   VAR_IN_OUT
      iqUDT_EquipmentControl : "UDT_EquipmentControl";   // Equipment control structure
      iqUDT_ConveyorInterface : "UDT_ConveyorInterface";   // Interface structure
   END_VAR

   VAR
      sx_EncoderFault { ExternalAccessible := 'False'; ExternalVisible := 'False'; ExternalWritable := 'False'} : Bool;   // When TRUE encoder fault is active
      slr_ActualDelayTime { ExternalAccessible := 'False'; ExternalVisible := 'False'; ExternalWritable := 'False'} : LReal;   // Actual delay time [ms]
   END_VAR

   VAR CONSTANT
      cudi_EncoderFaultDelayTime : UDInt := 5000;   // Time after which the encoder fault is activated
   END_VAR


BEGIN
	(*
	----------------------------------------------------------------------------------------

	Version history:
	Date        | Version   | Author        | Remark
	----------------------------------------------------------------------------------------
	19/07/2022  | 0.1       | M.Kurpiers    | first release MHS TIA 16.0
	21/02/2023  | 4.0       | F.Baten       | 4.0 Release TIA 17.5
	*)

	REGION 1 - Reset encoder error

	    IF #iqUDT_EquipmentControl.Command.Reset OR #iqUDT_ConveyorInterface.InternalErrorReset THEN
	        #sx_EncoderFault := FALSE;
	    END_IF;

	END_REGION

	REGION 2 - Set encoder error

	    IF #iqUDT_ConveyorInterface.ActualSpeed > 0
	        AND NOT #ix_EncoderPulses
	        AND NOT #iqUDT_ConveyorInterface.ManualModeActive THEN

	        #slr_ActualDelayTime += "DB_Memory".PrevCycleTime;

	        IF #slr_ActualDelayTime >= #cudi_EncoderFaultDelayTime THEN
	            #sx_EncoderFault := TRUE;
	        END_IF;
	    ELSE
	        #slr_ActualDelayTime := 0;
	    END_IF;

	    #iqUDT_ConveyorInterface.InternalErrorEncoder := #sx_EncoderFault;

	END_REGION

	REGION 3 - Status

	    #qUDT_HMIStatus.Fault := #sx_EncoderFault;

	END_REGION


END_FUNCTION_BLOCK

FUNCTION_BLOCK "FB_Valve"
TITLE = Single ended Valve Control and monitor
{ S7_Optimized_Access := 'TRUE' }
AUTHOR : 'I.Ajram'
VERSION : 0.1
   VAR_INPUT
      iUDT_Configuration { ExternalAccessible := 'False'; ExternalVisible := 'False'; ExternalWritable := 'False'} : "UDT_ValveConfiguration";   // Valve configuration
      ix_Open { ExternalAccessible := 'False'; ExternalVisible := 'False'; ExternalWritable := 'False'} : Bool;   // Open command (Hold if ControlMode = 1, pulse if ControlMode = 2)
      ix_Close { ExternalAccessible := 'False'; ExternalVisible := 'False'; ExternalWritable := 'False'} : Bool;   // Close command (Not used if ControlMode = 1, pulse if ControlMode = 2)
      ix_IsOpened { ExternalAccessible := 'False'; ExternalVisible := 'False'; ExternalWritable := 'False'} : Bool;   // Feedback Signal ( Not used if #iqUDT_SEVConfiguration.IsOpenFeedBackExist is FALSE)
      ix_IsClosed { ExternalAccessible := 'False'; ExternalVisible := 'False'; ExternalWritable := 'False'} : Bool;   // Feedback Signal ( Not used if #iqUDT_SEVConfiguration.IsCloseFeedBackExist is FALSE)
      ix_AirPressureOk { ExternalAccessible := 'False'; ExternalVisible := 'False'; ExternalWritable := 'False'} : Bool;   // Air pressure is healthy
   END_VAR

   VAR_OUTPUT
      qx_Open { ExternalAccessible := 'False'; ExternalVisible := 'False'; ExternalWritable := 'False'} : Bool;   // Open command
      qx_Close { ExternalAccessible := 'False'; ExternalVisible := 'False'; ExternalWritable := 'False'} : Bool;   // Close command
      qUDT_HMIStatus { ExternalAccessible := 'False'; ExternalVisible := 'False'; ExternalWritable := 'False'} : "UDT_ValveStatus";
      qUDT_Statistics { ExternalAccessible := 'False'; ExternalVisible := 'False'; ExternalWritable := 'False'} : "UDT_ValveStatistics";
   END_VAR

   VAR_IN_OUT
      iqUDT_HMICommand : "UDT_ValveCommand";   // Interafce for HMI commands
      iqUDT_Interface : "UDT_ValveInterface";   // Interface with external modules
      iqUDT_EquipmentControl : "UDT_EquipmentControl";   // Equipment control structure
   END_VAR

   VAR
      sx_ManualModeSelected { ExternalAccessible := 'False'; ExternalVisible := 'False'; ExternalWritable := 'False'} : Bool;
      sx_AutoModeSelected { ExternalAccessible := 'False'; ExternalVisible := 'False'; ExternalWritable := 'False'} : Bool;
      sx_OpenActivated { ExternalAccessible := 'False'; ExternalVisible := 'False'; ExternalWritable := 'False'} : Bool;
      sx_CloseActivated { ExternalAccessible := 'False'; ExternalVisible := 'False'; ExternalWritable := 'False'} : Bool;
      sx_FaultActive { ExternalAccessible := 'False'; ExternalVisible := 'False'; ExternalWritable := 'False'} : Bool;
      sTON_Opening {InstructionName := 'TON_TIME'; LibVersion := '1.0'; ExternalAccessible := 'False'; ExternalVisible := 'False'; ExternalWritable := 'False'; S7_SetPoint := 'False'} : TON_TIME;
      sTON_Closing {InstructionName := 'TON_TIME'; LibVersion := '1.0'; ExternalAccessible := 'False'; ExternalVisible := 'False'; ExternalWritable := 'False'; S7_SetPoint := 'False'} : TON_TIME;
      sTime_Closing { ExternalAccessible := 'False'; ExternalVisible := 'False'; ExternalWritable := 'False'} : Time;
      sTime_Opening { ExternalAccessible := 'False'; ExternalVisible := 'False'; ExternalWritable := 'False'} : Time;
      RTRIG_Open {InstructionName := 'R_TRIG'; LibVersion := '1.0'; ExternalAccessible := 'False'; ExternalVisible := 'False'; ExternalWritable := 'False'; S7_SetPoint := 'False'} : R_TRIG;
      RTRIG_Close {InstructionName := 'R_TRIG'; LibVersion := '1.0'; ExternalAccessible := 'False'; ExternalVisible := 'False'; ExternalWritable := 'False'; S7_SetPoint := 'False'} : R_TRIG;
      RTRIG_FaultActive {InstructionName := 'R_TRIG'; LibVersion := '1.0'; ExternalAccessible := 'False'; ExternalVisible := 'False'; ExternalWritable := 'False'; S7_SetPoint := 'False'} : R_TRIG;
      RTRIG_Opened {InstructionName := 'R_TRIG'; LibVersion := '1.0'; ExternalAccessible := 'False'; ExternalVisible := 'False'; ExternalWritable := 'False'; S7_SetPoint := 'False'} : R_TRIG;
   END_VAR

   VAR CONSTANT
      ci_ControlModeHold : Int := 1;   // Energize to hold
      ci_ControlModePulse : Int := 2;   // Pulse energized to change state
      ci_ValveTypeSEV : Int := 1;   // Single coil valve
      ci_ValveTypeDEV : Int := 2;   // Double coil valve, bi-stable, latching
   END_VAR


BEGIN
	(*
	----------------------------------------------------------------------------------------

	Version history:
	Date        | Version   | Author        | Remark
	----------------------------------------------------------------------------------------
	08/07/2024  | 0.1       | I. Ajram      | first release TIA 18
	16/07/2024  | 0.2       | I. Ajram      | Changed block name from FB_SEV to FB_Valve
	                                        |  +    Added Configuration to allow for SEV and DEV
	                                        |  +    Added qx_Close Output
	                                        |  +    Added logic to accomodate for DEV
	30/08/2024  | 0.3       | J. Majer      | Added comments, number regions, added iq_UDT_EquipmentInterface, iqUDT_EquipmentControl
	----------------------------------------------------------------------------------------

	*)

	REGION 1 - Edge detection
	    // Trigger rising edge detection for different signals: Open, Close, FaultActive, and Opened.
	    #RTRIG_Open(CLK := #ix_Open OR #iqUDT_Interface.Open);
	    #RTRIG_Close(CLK := #ix_Close OR #iqUDT_Interface.Close);
	    #RTRIG_FaultActive(CLK := #sx_FaultActive);
	    #RTRIG_Opened(CLK := #qUDT_HMIStatus.Specific.Opened);

	END_REGION

	REGION 2 - Auto / Manual

	    // Handle auto mode command.
	    IF #iqUDT_EquipmentControl.Command.Start AND #iqUDT_EquipmentControl.Command.AutomaticOn
	    THEN
	        #sx_AutoModeSelected := TRUE;
	        #sx_ManualModeSelected := FALSE;
	        #iqUDT_HMICommand.AutoMode := FALSE;
	    END_IF;

	    // Manual mode bits inputs can be reset in case of malfunction
	    IF #iqUDT_EquipmentControl.Command.DisableManualMode
	    THEN
	        #iqUDT_HMICommand.ManualMode := FALSE;
	        #iqUDT_EquipmentControl.Command.ManualMode := FALSE;
	    END_IF;

	    // Handle manual mode command.
	    IF (#iqUDT_EquipmentControl.Command.ManualMode OR #iqUDT_HMICommand.ManualMode)
	        AND NOT #iqUDT_EquipmentControl.Command.DisableManualMode
	    THEN
	        #sx_AutoModeSelected := FALSE;
	        #sx_ManualModeSelected := TRUE;
	        #iqUDT_HMICommand.ManualMode := FALSE;
	    END_IF;

	    REGION 2.1 - Restart request

	        // Indicating need for system restart if no mode is selected
	        #iqUDT_EquipmentControl.Request.RestartRequired := NOT #sx_AutoModeSelected
	        AND NOT #sx_AutoModeSelected;

	    END_REGION
	END_REGION

	REGION 3 - Faults

	    REGION 3.1 - Configuration Error
	        // Check for configuration errors by validating the ControlMode and ValveType values.
	        IF #iUDT_Configuration.ControlMode < #ci_ControlModeHold
	            OR #iUDT_Configuration.ControlMode > #ci_ControlModePulse
	            OR #iUDT_Configuration.ValveType < #ci_ValveTypeSEV
	            OR #iUDT_Configuration.ValveType > #ci_ValveTypeDEV
	        THEN
	            #qUDT_HMIStatus.Specific.ConfigurationError := TRUE;
	        ELSE
	            #qUDT_HMIStatus.Specific.ConfigurationError := FALSE;
	        END_IF;

	    END_REGION

	    REGION 3.2 - Low Pressure
	        // Set AirPressureLost flag if air pressure is not okay.
	        IF NOT #ix_AirPressureOk THEN
	            #qUDT_HMIStatus.Specific.AirPressureLost := TRUE;
	        END_IF;

	    END_REGION

	    REGION 3.3 - Fail to Open
	        // Set FailToOpen flag if the valve failed to open within the expected time.
	        IF #sTON_Opening.Q AND #iUDT_Configuration.OpenFeedBackExist THEN
	            #qUDT_HMIStatus.Specific.FailToOpen := TRUE;
	        END_IF;

	    END_REGION

	    REGION 3.4 - Fail to Close
	        // Set FailToClose flag if the valve failed to close within the expected time.
	        IF #sTON_Closing.Q AND #iUDT_Configuration.CloseFeedBackExist THEN
	            #qUDT_HMIStatus.Specific.FailToClose := TRUE;
	        END_IF;

	    END_REGION

	    REGION 3.4 - Collective fault
	        // Set FaultActive flag if any specific fault is detected (fail to open/close, air pressure lost, or configuration error).
	        #sx_FaultActive := #qUDT_HMIStatus.Specific.FailToClose OR
	        #qUDT_HMIStatus.Specific.FailToOpen OR
	        #qUDT_HMIStatus.Specific.AirPressureLost OR
	        #qUDT_HMIStatus.Specific.ConfigurationError;

	        // forward error to the interface with other modules
	        #iqUDT_Interface.Error := #sx_FaultActive;

	        // If FaultActive is set, deactivate open and close commands.
	        IF #sx_FaultActive THEN
	            #sx_OpenActivated := FALSE;
	            #sx_CloseActivated := FALSE;
	        END_IF;

	    END_REGION

	    REGION 3.5 - Reset
	        // Reset fault flags and set air pressure flag based on the state of AirPressureOk.
	        IF #iqUDT_EquipmentControl.Command.Reset THEN
	            #qUDT_HMIStatus.Specific.FailToOpen := FALSE;
	            #qUDT_HMIStatus.Specific.FailToClose := FALSE;
	            #qUDT_HMIStatus.Specific.AirPressureLost := NOT #ix_AirPressureOk;
	        END_IF;

	    END_REGION

	END_REGION

	REGION 4 - Command
	    // Process commands based on the current mode (Auto/Manual) and fault state.
	    IF NOT #sx_FaultActive THEN

	        REGION 4.1 - Auto
	            // Handle command logic in Auto mode based on control mode (Hold or Pulse).
	            IF #sx_AutoModeSelected THEN
	                CASE #iUDT_Configuration.ControlMode OF

	                        // ControlModeHold: Open/close based on the ix_Open signal.
	                    #ci_ControlModeHold:
	                        #sx_OpenActivated := #ix_Open;
	                        #sx_CloseActivated := NOT #ix_Open;

	                        // ControlModePulse: Open/close based on rising edge detection.
	                    #ci_ControlModePulse:
	                        IF #RTRIG_Open.Q AND NOT #ix_IsOpened THEN
	                            #sx_OpenActivated := TRUE;
	                            #sx_CloseActivated := FALSE;
	                        END_IF;

	                        IF #RTRIG_Close.Q AND NOT #ix_IsClosed THEN
	                            #sx_OpenActivated := FALSE;
	                            #sx_CloseActivated := TRUE;
	                        END_IF;

	                END_CASE;
	            END_IF;

	        END_REGION

	        REGION 4.2 - Manual
	            // Handle command logic in Manual mode based on control mode (Hold or Pulse).
	            IF #sx_ManualModeSelected THEN
	                CASE #iUDT_Configuration.ControlMode OF

	                        // ControlModeHold: Open/close based on manual commands.
	                    #ci_ControlModeHold:
	                        #sx_OpenActivated := #iqUDT_HMICommand.ManualOpen;
	                        #sx_CloseActivated := #iqUDT_HMICommand.ManualClose;

	                        // ControlModePulse: Open/close based on manual commands with feedback checks.
	                    #ci_ControlModePulse:
	                        IF #iqUDT_HMICommand.ManualOpen AND NOT #ix_IsOpened THEN
	                            #sx_OpenActivated := TRUE;
	                            #sx_CloseActivated := FALSE;
	                            #iqUDT_HMICommand.ManualOpen := FALSE;
	                        END_IF;

	                        IF #iqUDT_HMICommand.ManualClose AND NOT #ix_IsClosed THEN
	                            #sx_OpenActivated := FALSE;
	                            #sx_CloseActivated := TRUE;
	                            #iqUDT_HMICommand.ManualClose := FALSE;
	                        END_IF;

	                END_CASE;
	            END_IF;

	        END_REGION
	    ELSE
	        // On fault, clear all open/close commands.
	        #sx_OpenActivated := FALSE;
	        #sx_CloseActivated := FALSE;
	        #iqUDT_HMICommand.ManualClose := FALSE;
	        #iqUDT_HMICommand.ManualOpen := FALSE;
	    END_IF;

	END_REGION

	REGION 5 - Statistics
	    // Update statistical data when reset or fault occurs.
	    IF #iqUDT_EquipmentControl.Command.ResetData OR #sx_FaultActive THEN
	        "FC_Statistics"(ix_Reset := #iqUDT_EquipmentControl.Command.ResetData,
	                        ix_Activate := #sx_FaultActive,
	                        ix_RTrigActivate := #RTRIG_FaultActive.Q,
	                        iqUDT_Statistics := #qUDT_Statistics.Fail);
	    END_IF;

	    // Update open statistics when reset or opened.
	    IF #iqUDT_EquipmentControl.Command.ResetData OR #qUDT_HMIStatus.Specific.Opened THEN
	        "FC_Statistics"(ix_Reset := #iqUDT_EquipmentControl.Command.ResetData,
	                        ix_Activate := #qUDT_HMIStatus.Specific.Opened,
	                        ix_RTrigActivate := #RTRIG_Opened.Q,
	                        iqUDT_Statistics := #qUDT_Statistics.Open);
	    END_IF;

	END_REGION

	REGION 6 - Status

	    REGION 6.1 - Opened / Closed
	        // Handle open/close status based on feedback or timers.
	        IF #iUDT_Configuration.OpenFeedBackExist THEN
	            // Set opened status based on feedback.
	            #qUDT_HMIStatus.Specific.Opened := #ix_IsOpened;
	        ELSE
	            // Use opening timer as an indicator if feedback is not available.
	            IF #sTON_Opening.Q THEN
	                #qUDT_HMIStatus.Specific.Opened := TRUE;
	            END_IF;
	            IF #sx_CloseActivated THEN
	                #qUDT_HMIStatus.Specific.Opened := FALSE;
	            END_IF;
	        END_IF;

	        // Module interface valve feedback opened
	        #iqUDT_Interface.IsOpened := #qUDT_HMIStatus.Specific.Opened;

	        IF #iUDT_Configuration.CloseFeedBackExist THEN
	            // Set closed status based on feedback.
	            #qUDT_HMIStatus.Specific.Closed := #ix_IsClosed;
	        ELSE
	            // Use closing timer as an indicator if feedback is not available.
	            IF #sTON_Closing.Q THEN
	                #qUDT_HMIStatus.Specific.Closed := TRUE;
	            END_IF;
	            IF #sx_OpenActivated THEN
	                #qUDT_HMIStatus.Specific.Closed := FALSE;
	            END_IF;
	        END_IF;

	        // Module interface valve feedback closed
	        #iqUDT_Interface.IsClosed := #qUDT_HMIStatus.Specific.Closed;

	    END_REGION

	    REGION 6.2 - Opening
	        // Handle the logic for the valve opening, including timer initialization and status updates.
	        IF #iUDT_Configuration.OpenTime = 0 THEN
	            #sTime_Opening := T#1s;  // Default to 1 second if not configured.
	        ELSE
	            #sTime_Opening := INT_TO_TIME(#iUDT_Configuration.OpenTime);  // Use configured open time.
	        END_IF;

	        IF #sx_OpenActivated AND NOT #qUDT_HMIStatus.Specific.Opened THEN
	            #qUDT_HMIStatus.Specific.Opening := TRUE;
	        ELSE
	            #qUDT_HMIStatus.Specific.Opening := FALSE;
	        END_IF;

	        // Start the opening timer.
	        #sTON_Opening(IN := #qUDT_HMIStatus.Specific.Opening,
	                      PT := #sTime_Opening);

	    END_REGION

	    REGION 6.3 - Closing
	        // Handle the logic for the valve closing, including timer initialization and status updates.
	        IF #iUDT_Configuration.CloseTime = 0 THEN
	            #sTime_Closing := T#1s;  // Default to 1 second if not configured.
	        ELSE
	            #sTime_Closing := INT_TO_TIME(#iUDT_Configuration.CloseTime);  // Use configured close time.
	        END_IF;

	        IF #sx_CloseActivated AND NOT #qUDT_HMIStatus.Specific.Closed THEN
	            #qUDT_HMIStatus.Specific.Closing := TRUE;
	        ELSE
	            #qUDT_HMIStatus.Specific.Closing := FALSE;
	        END_IF;

	        // Start the closing timer.
	        #sTON_Closing(IN := #qUDT_HMIStatus.Specific.Closing,
	                      PT := #sTime_Closing);

	    END_REGION

	END_REGION

	REGION 7 - Output

	    // Select the action based on the valve type configuration
	    CASE #iUDT_Configuration.ValveType OF

	            // SEV Valve Type
	        #ci_ValveTypeSEV:
	            // The valve opens if Open is activated, Close is not activated, and no fault is active
	            #qx_Open :=
	            #sx_OpenActivated AND
	            NOT #sx_CloseActivated AND
	            NOT #sx_FaultActive;

	            // Reset the open signal, SEV logic requires manual reset after operation
	            #qx_Open := FALSE;

	            // DEV Valve Type
	        #ci_ValveTypeDEV:
	            // The valve opens if there are no faults, Open is activated, and the valve is not yet opened
	            #qx_Open :=
	            NOT #sx_FaultActive AND
	            #sx_OpenActivated AND NOT #qUDT_HMIStatus.Specific.Opened;

	            // The valve closes if there are no faults, Close is activated, and the valve is not yet closed
	            #qx_Close :=
	            NOT #sx_FaultActive AND
	            #sx_CloseActivated AND NOT #qUDT_HMIStatus.Specific.Closed;

	            // If the valve is opened, a fault occurs, or the valve is in the closing state, deactivate Open
	            IF #qUDT_HMIStatus.Specific.Opened OR
	                #sx_FaultActive OR
	                #qUDT_HMIStatus.Specific.Closing
	            THEN
	                #sx_OpenActivated := FALSE;
	            END_IF;

	            // If the valve is closed, a fault occurs, or the valve is in the opening state, deactivate Close
	            IF #qUDT_HMIStatus.Specific.Closed OR
	                #sx_FaultActive OR
	                #qUDT_HMIStatus.Specific.Opening
	            THEN
	                #sx_CloseActivated := FALSE;
	            END_IF;

	    END_CASE;

	END_REGION

END_FUNCTION_BLOCK

FUNCTION_BLOCK "FB_ConveyorPanel"
{ S7_Optimized_Access := 'TRUE' }
AUTHOR : MHSE
VERSION : 3.0
// ATTRIBUTES
// AUTO_NUMBER = True
// BLOCK_NUMBER = 6
// END_ATTRIBUTES
//Main switch and 24V feeedback available in VFD cabinet
   VAR_INPUT
      ix_MainSwitchOk { ExternalAccessible := 'False'; ExternalVisible := 'False'; ExternalWritable := 'False'} : Bool;   // TRUE if main switch with no fault
      ix_CBFeedback { ExternalAccessible := 'False'; ExternalVisible := 'False'; ExternalWritable := 'False'} : Bool;   // TRUE if circuit breacker is ON
      ix_HardwareOk { ExternalAccessible := 'False'; ExternalVisible := 'False'; ExternalWritable := 'False'} : Bool;   // TRUE when hardware is Ok
   END_VAR

   VAR_OUTPUT
      qUDT_HMIStatus { ExternalAccessible := 'False'; ExternalVisible := 'False'; ExternalWritable := 'False'} : "UDT_ConveyorPanelStatus";   // HMI status structure
   END_VAR

   VAR_IN_OUT
      iqUDT_ConveyorInterface : "UDT_ConveyorInterface";   // Conveyor interface structure
      iqUDT_Statistics : "UDT_ConveyorPanelStatistics";   // Statistics structure
   END_VAR

   VAR
      sUDT_HMIStatus { ExternalAccessible := 'False'; ExternalVisible := 'False'; ExternalWritable := 'False'; S7_SetPoint := 'False'} : "UDT_ConveyorPanelStatus";   // Conveyor Panel status UDT
      sR_Trig_24VDC {InstructionName := 'R_TRIG'; LibVersion := '1.0'; ExternalAccessible := 'False'; ExternalVisible := 'False'; ExternalWritable := 'False'; S7_SetPoint := 'False'} : R_TRIG;   // Rise trigger when a 24VDC fault occurs
      sR_Trig_MainSwitch {InstructionName := 'R_TRIG'; LibVersion := '1.0'; ExternalAccessible := 'False'; ExternalVisible := 'False'; ExternalWritable := 'False'; S7_SetPoint := 'False'} : R_TRIG;   // Rise trigger when a Main switch fault occurs
   END_VAR


BEGIN
	(*
	----------------------------------------------------------------------------------------

	Version history:
	Date        | Version   | Author        | Remark
	----------------------------------------------------------------------------------------
	10/01/2020  | 3.0       | S. Nikodem    | first release MHS TIA 15.1
	16/10/2020  | 3.1       | S. Deulkar    | Changed 24VDc input name to CBFeedback, also UDT are updated
	21/02/2023  | 4.0       | F.Baten       | 4.0 Release TIA 17.5
	*)

	REGION 1 - Triggers

	    // Rise trigger 24VDC status
	    #sR_Trig_24VDC(CLK := #sUDT_HMIStatus.CBFeedbackError);

	    // Rise trigger Main switch status
	    #sR_Trig_MainSwitch(CLK := #sUDT_HMIStatus.MainSwitchOff);

	END_REGION

	REGION 2 - Reset error

	    IF #iqUDT_ConveyorInterface.InternalErrorReset
	    THEN

	        #sUDT_HMIStatus.CBFeedbackError := FALSE;
	        #sUDT_HMIStatus.MainSwitchOff := FALSE;

	    END_IF;

	END_REGION

	REGION 3 - Faults monitoring

	    // 24 VDC fault status is set when the 24V error occurred
	    IF NOT #ix_CBFeedback
	    THEN

	        #sUDT_HMIStatus.CBFeedbackError := TRUE;

	    END_IF;

	    // Main switch fault status is set when the main switch error occurred
	    IF NOT #ix_MainSwitchOk
	    THEN

	        #sUDT_HMIStatus.MainSwitchOff := TRUE;

	    END_IF;

	    // Set disconnect bit on Conveyor interface
	    #iqUDT_ConveyorInterface.Disconnected := #sUDT_HMIStatus.CBFeedbackError OR #sUDT_HMIStatus.MainSwitchOff;

	    // Move static structure to output
	    #qUDT_HMIStatus := #sUDT_HMIStatus;

	END_REGION

	REGION 4 - Statistics

	    // 24 VDC Supply fault statistics

	    IF #sUDT_HMIStatus.CBFeedbackError
	        OR #iqUDT_ConveyorInterface.ResetStatistics
	    THEN

	        "FC_Statistics"(ix_Reset := #iqUDT_ConveyorInterface.ResetStatistics,
	                        ix_Activate := #sUDT_HMIStatus.CBFeedbackError,
	                        ix_RTrigActivate := #sR_Trig_24VDC.Q,
	                        iqUDT_Statistics := #iqUDT_Statistics.CBFeedbackError);

	    END_IF;

	    // Main switch fault statistics

	    IF #sUDT_HMIStatus.MainSwitchOff
	        OR #iqUDT_ConveyorInterface.ResetStatistics
	    THEN

	        "FC_Statistics"(ix_Reset := #iqUDT_ConveyorInterface.ResetStatistics,
	                        ix_Activate := #sUDT_HMIStatus.MainSwitchOff,
	                        ix_RTrigActivate := #sR_Trig_MainSwitch.Q,
	                        iqUDT_Statistics := #iqUDT_Statistics.MainSwitchOff);

	    END_IF;

	END_REGION

END_FUNCTION_BLOCK

FUNCTION_BLOCK "FB_ConvertGIN"
{ S7_Optimized_Access := 'TRUE' }
VERSION : 0.1
// ATTRIBUTES
// AUTO_NUMBER = True
// BLOCK_NUMBER = 5
// END_ATTRIBUTES
   VAR_INPUT
      ii_GINRangeStart { ExternalAccessible := 'False'; ExternalVisible := 'False'; ExternalWritable := 'False'} : Int;   // GIN range start
      ii_GINRangeEnd { ExternalAccessible := 'False'; ExternalVisible := 'False'; ExternalWritable := 'False'} : Int;   // GIN range end
   END_VAR

   VAR_IN_OUT
      iqUDT_Handshake : "UDT_ConveyorHandshake";   // Conveyor handshake structure
      iqUDT_UnknownGIN : "UDT_UnknownGIN";   // Unknown GIN structure
   END_VAR

   VAR
      sR_TRIG_NewGINDetected {InstructionName := 'R_TRIG'; LibVersion := '1.0'; ExternalAccessible := 'False'; ExternalVisible := 'False'; ExternalWritable := 'False'; S7_SetPoint := 'False'} : R_TRIG;   // New GIN detected rising edge
      si_LastGenGIN { ExternalAccessible := 'False'; ExternalVisible := 'False'; ExternalWritable := 'False'} : Int;   // Last generated GIN
      si_GenGIN { ExternalAccessible := 'False'; ExternalVisible := 'False'; ExternalWritable := 'False'} : Int;   // Generated GIN
      si_DetectedGIN { ExternalAccessible := 'False'; ExternalVisible := 'False'; ExternalWritable := 'False'} : Int;   // Last detected GIN
      sx_GINOutOfRange { ExternalAccessible := 'False'; ExternalVisible := 'False'; ExternalWritable := 'False'} : Bool;   // GIN out of range
   END_VAR


BEGIN
	(*
	----------------------------------------------------------------------------------------

	Version history:
	Date        | Version   | Author        | Remark
	----------------------------------------------------------------------------------------
	15/01/2020  | 3.0       | L.Klar        | first release MHS TIA 15.1
	03/03/2020  | 3.1       | P. Pielucha   | Adapting reviews
	21/02/2023  | 4.0       | F.Baten       | 4.0 Release TIA 17.5
	*)

	REGION 1 – GIN generator initialization

	    // Initialize GIN if last generated GIN is out of configured range.
	    IF (#si_LastGenGIN < #ii_GINRangeStart
	        OR #si_LastGenGIN > #ii_GINRangeEnd)
	    THEN

	        #si_LastGenGIN := #ii_GINRangeStart - 1;

	    END_IF;

	END_REGION

	REGION 2 – GIN conversion

	    // Riding edge on new GIN detected
	    #sR_TRIG_NewGINDetected(CLK := #iqUDT_Handshake.GIN > 0 AND #iqUDT_Handshake.GIN <> #si_DetectedGIN);

	    // Check if detected GIN is out of normal and unknown GIN ranges
	    #sx_GINOutOfRange := (#iqUDT_Handshake.GIN < #ii_GINRangeStart
	    OR #iqUDT_Handshake.GIN > #ii_GINRangeEnd)
	    AND (#iqUDT_Handshake.GIN < #iqUDT_UnknownGIN.Start OR
	    #iqUDT_Handshake.GIN > #iqUDT_UnknownGIN.End);

	    // Generate new GIN if new GIN was detected
	    IF (#sR_TRIG_NewGINDetected.Q
	        AND #sx_GINOutOfRange)
	    THEN

	        #si_DetectedGIN := #iqUDT_Handshake.GIN;

	        IF (#si_LastGenGIN < #ii_GINRangeEnd)
	        THEN

	            #si_GenGIN := #si_LastGenGIN + 1;
	            #si_LastGenGIN += 1;

	        ELSE

	            #si_GenGIN := #ii_GINRangeStart;
	            #si_LastGenGIN := #ii_GINRangeStart;

	        END_IF;

	        // Copy detected GIN record to new generated GIN
	        "DB_GIN".GIN[#si_GenGIN] := "DB_GIN".GIN[#si_DetectedGIN];

	    END_IF;

	    // GIN update
	    IF (#iqUDT_Handshake.GIN > 0
	        AND #sx_GINOutOfRange)
	    THEN

	        #iqUDT_Handshake.GIN := #si_GenGIN;

	    END_IF;

	END_REGION
END_FUNCTION_BLOCK

FUNCTION_BLOCK "FB_GapOptimizationSystem"
{ S7_Optimized_Access := 'TRUE' }
VERSION : 0.1
// ATTRIBUTES
// AUTO_NUMBER = True
// BLOCK_NUMBER = 9
// END_ATTRIBUTES
   VAR_INPUT
      iUDT_GOSConfiguration { ExternalAccessible := 'False'; ExternalVisible := 'False'; ExternalWritable := 'False'} : "UDT_GapOptimizationSystemConfiguration";   // UDT of the Gap Optimization System Configuration
      iUDT_ConvA { ExternalAccessible := 'False'; ExternalVisible := 'False'; ExternalWritable := 'False'} : "UDT_ConveyorInterface";
      iUDT_ConvB { ExternalAccessible := 'False'; ExternalVisible := 'False'; ExternalWritable := 'False'} : "UDT_ConveyorInterface";
      iUDT_ConvC { ExternalAccessible := 'False'; ExternalVisible := 'False'; ExternalWritable := 'False'} : "UDT_ConveyorInterface";
      iUDT_ConvUpstream { ExternalAccessible := 'False'; ExternalVisible := 'False'; ExternalWritable := 'False'} : "UDT_ConveyorInterface";
      iUDT_HandshakeUp { ExternalAccessible := 'False'; ExternalVisible := 'False'; ExternalWritable := 'False'} : "UDT_ConveyorHandshake";
      ii_LoopSpeed { ExternalAccessible := 'False'; ExternalVisible := 'False'; ExternalWritable := 'False'} : Int := 2900;   // Set Speed of Loop conveyors
      ix_PECUpstream { ExternalAccessible := 'False'; ExternalVisible := 'False'; ExternalWritable := 'False'} : Bool;
      ix_PECA1 { ExternalAccessible := 'False'; ExternalVisible := 'False'; ExternalWritable := 'False'} : Bool;   // BOS PEC of conveyor A
      ix_PECA2 { ExternalAccessible := 'False'; ExternalVisible := 'False'; ExternalWritable := 'False'} : Bool;   // EOS PEC of conveyor A
      ix_PECB1 { ExternalAccessible := 'False'; ExternalVisible := 'False'; ExternalWritable := 'False'} : Bool;   // BOS PEC of conveyor B
      ix_PECB2 { ExternalAccessible := 'False'; ExternalVisible := 'False'; ExternalWritable := 'False'} : Bool;   // EOS PEC of conveyor B
      ix_PECC1 { ExternalAccessible := 'False'; ExternalVisible := 'False'; ExternalWritable := 'False'} : Bool;   // BOS PEC of conveyor C
      ix_PECC2 { ExternalAccessible := 'False'; ExternalVisible := 'False'; ExternalWritable := 'False'} : Bool;   // EOS PEC of conveyor C
      ix_PECDownstream { ExternalAccessible := 'False'; ExternalVisible := 'False'; ExternalWritable := 'False'} : Bool;
   END_VAR

   VAR_OUTPUT
      qUDT_GOSStatus { ExternalAccessible := 'False'; ExternalVisible := 'False'; ExternalWritable := 'False'} : "UDT_GapOptimizationSystemStatus";   // UDT of the Gap Optimization System Status
   END_VAR

   VAR_IN_OUT
      iqUDT_GOSInterface : "UDT_GapOptimizationSystemInterface";   // UDT of the Gap Optimization System Interface
      iqUDT_GOSLog : Array[*] of "UDT_GOSLog";
      iqa_TrackingDataUpstream : Array[*] of Int;   // Tracking data of the upstream conveyor
      iqa_TrackingDataA : Array[*] of Int;   // Tracking data of conveyor A
      iqa_TrackingDataB : Array[*] of Int;   // Tracking data of conveyor B
      iqa_TrackingDataC : Array[*] of Int;   // Tracking data of conveyor C
      iqa_TrackingDataDownstream : Array[*] of Int;   // Tracking data of the downstream conveyor
      iqx_ShiftRequest { ExternalAccessible := 'False'; ExternalVisible := 'False'; ExternalWritable := 'False'} : Bool;   // Request to Shift
   END_VAR

   VAR
      sr_TravelDistanceUpstreamParc { ExternalAccessible := 'False'; ExternalVisible := 'False'; ExternalWritable := 'False'} : Real;   // Travel distance of the upstream parcel (mm)
      sr_TravelDistanceCurrentParcA { ExternalAccessible := 'False'; ExternalVisible := 'False'; ExternalWritable := 'False'} : Real;   // Travel distance of the current parcel on Conv. A (mm)
      sr_TravelDistanceUpstreamParcA { ExternalAccessible := 'False'; ExternalVisible := 'False'; ExternalWritable := 'False'} : Real;   // Travel distance of the upstream parcel before it reaches Conv. A (mm)
      sr_TravelDistanceCurrentParcB { ExternalAccessible := 'False'; ExternalVisible := 'False'; ExternalWritable := 'False'} : Real;   // Travel distance of the current parcel on Conv. B (mm)
      sr_TravelDistanceUpstreamParcB { ExternalAccessible := 'False'; ExternalVisible := 'False'; ExternalWritable := 'False'} : Real;   // Travel distance of the upstream parcel before it reaches Conv. B (mm)
      sr_TravelDistanceCurrentParcC { ExternalAccessible := 'False'; ExternalVisible := 'False'; ExternalWritable := 'False'} : Real;   // Travel distance of the current parcel on Conv. C (mm)
      sa_ParcelA1 { ExternalAccessible := 'False'; ExternalVisible := 'False'; ExternalWritable := 'False'} : Struct   // Struct of a parcel
         GIN { ExternalAccessible := 'False'; ExternalVisible := 'False'; ExternalWritable := 'False'} : Int;   // GIN number
         Length { ExternalAccessible := 'False'; ExternalVisible := 'False'; ExternalWritable := 'False'} : Int;   // Length current parcel (mm)
         GapUpstream { ExternalAccessible := 'False'; ExternalVisible := 'False'; ExternalWritable := 'False'} : Int;   // Length of the gap upstream (mm)
         GapDownstream { ExternalAccessible := 'False'; ExternalVisible := 'False'; ExternalWritable := 'False'} : Int;   // Length of the gap downstream (mm)
         GapToBeRecovered { ExternalAccessible := 'False'; ExternalVisible := 'False'; ExternalWritable := 'False'} : Int;   // Length of the recovered gap (mm)
         GapCovered { ExternalAccessible := 'False'; ExternalVisible := 'False'; ExternalWritable := 'False'} : Int;   // Length of  the covered gap (mm)
         LogNr { ExternalAccessible := 'False'; ExternalVisible := 'False'; ExternalWritable := 'False'} : Int;
         Accelerate { ExternalAccessible := 'False'; ExternalVisible := 'False'; ExternalWritable := 'False'} : Bool;   // True is acceleration needed
         Decelerate { ExternalAccessible := 'False'; ExternalVisible := 'False'; ExternalWritable := 'False'} : Bool;   // True is deceleration needed
      END_STRUCT;
      sa_ParcelB1 { ExternalAccessible := 'False'; ExternalVisible := 'False'; ExternalWritable := 'False'} : Struct   // Struct of a parcel
         GIN { ExternalAccessible := 'False'; ExternalVisible := 'False'; ExternalWritable := 'False'} : Int;   // GIN number
         Length { ExternalAccessible := 'False'; ExternalVisible := 'False'; ExternalWritable := 'False'} : Int;   // Length current parcel (mm)
         GapUpstream { ExternalAccessible := 'False'; ExternalVisible := 'False'; ExternalWritable := 'False'} : Int;   // Length of the gap upstream (mm)
         GapDownstream { ExternalAccessible := 'False'; ExternalVisible := 'False'; ExternalWritable := 'False'} : Int;   // Length of the gap downstream (mm)
         GapToBeRecovered { ExternalAccessible := 'False'; ExternalVisible := 'False'; ExternalWritable := 'False'} : Int;   // Length of the recovered gap (mm)
         GapCovered { ExternalAccessible := 'False'; ExternalVisible := 'False'; ExternalWritable := 'False'} : Int;   // Length of  the covered gap (mm)
         LogNr { ExternalAccessible := 'False'; ExternalVisible := 'False'; ExternalWritable := 'False'} : Int;
         Accelerate { ExternalAccessible := 'False'; ExternalVisible := 'False'; ExternalWritable := 'False'} : Bool;   // True is acceleration needed
         Decelerate { ExternalAccessible := 'False'; ExternalVisible := 'False'; ExternalWritable := 'False'} : Bool;   // True is deceleration needed
      END_STRUCT;
      sa_ParcelC1 { ExternalAccessible := 'False'; ExternalVisible := 'False'; ExternalWritable := 'False'} : Struct   // Struct of a parcel
         GIN { ExternalAccessible := 'False'; ExternalVisible := 'False'; ExternalWritable := 'False'} : Int;   // GIN number
         Length { ExternalAccessible := 'False'; ExternalVisible := 'False'; ExternalWritable := 'False'} : Int;   // Length current parcel (mm)
         GapUpstream { ExternalAccessible := 'False'; ExternalVisible := 'False'; ExternalWritable := 'False'} : Int;   // Length of the gap upstream (mm)
         GapDownstream { ExternalAccessible := 'False'; ExternalVisible := 'False'; ExternalWritable := 'False'} : Int;   // Length of the gap downstream (mm)
         GapToBeRecovered { ExternalAccessible := 'False'; ExternalVisible := 'False'; ExternalWritable := 'False'} : Int;   // Length of the recovered gap (mm)
         GapCovered { ExternalAccessible := 'False'; ExternalVisible := 'False'; ExternalWritable := 'False'} : Int;   // Length of  the covered gap (mm)
         LogNr { ExternalAccessible := 'False'; ExternalVisible := 'False'; ExternalWritable := 'False'} : Int;
         Accelerate { ExternalAccessible := 'False'; ExternalVisible := 'False'; ExternalWritable := 'False'} : Bool;   // True is acceleration needed
         Decelerate { ExternalAccessible := 'False'; ExternalVisible := 'False'; ExternalWritable := 'False'} : Bool;   // True is deceleration needed
      END_STRUCT;
      sa_ParcelC2 { ExternalAccessible := 'False'; ExternalVisible := 'False'; ExternalWritable := 'False'} : Struct   // Struct of a parcel
         GIN { ExternalAccessible := 'False'; ExternalVisible := 'False'; ExternalWritable := 'False'} : Int;   // GIN number
         Length { ExternalAccessible := 'False'; ExternalVisible := 'False'; ExternalWritable := 'False'} : Int;   // Length current parcel (mm)
         GapUpstream { ExternalAccessible := 'False'; ExternalVisible := 'False'; ExternalWritable := 'False'} : Int;   // Length of the gap upstream (mm)
         GapDownstream { ExternalAccessible := 'False'; ExternalVisible := 'False'; ExternalWritable := 'False'} : Int;   // Length of the gap downstream (mm)
         GapToBeRecovered { ExternalAccessible := 'False'; ExternalVisible := 'False'; ExternalWritable := 'False'} : Int;   // Length of the recovered gap (mm)
         GapCovered { ExternalAccessible := 'False'; ExternalVisible := 'False'; ExternalWritable := 'False'} : Int;   // Length of  the covered gap (mm)
         LogNr { ExternalAccessible := 'False'; ExternalVisible := 'False'; ExternalWritable := 'False'} : Int;
         Accelerate { ExternalAccessible := 'False'; ExternalVisible := 'False'; ExternalWritable := 'False'} : Bool;   // True is acceleration needed
         Decelerate { ExternalAccessible := 'False'; ExternalVisible := 'False'; ExternalWritable := 'False'} : Bool;   // True is deceleration needed
      END_STRUCT;
      ss_AnotherParcelatB { ExternalAccessible := 'False'; ExternalVisible := 'False'; ExternalWritable := 'False'} : Struct   // Struct of a parcel
         GIN { ExternalAccessible := 'False'; ExternalVisible := 'False'; ExternalWritable := 'False'} : Int;   // GIN number
         Length { ExternalAccessible := 'False'; ExternalVisible := 'False'; ExternalWritable := 'False'} : Int;   // Length current parcel (mm)
         GapUpstream { ExternalAccessible := 'False'; ExternalVisible := 'False'; ExternalWritable := 'False'} : Int;   // Length of the gap upstream (mm)
         GapDownstream { ExternalAccessible := 'False'; ExternalVisible := 'False'; ExternalWritable := 'False'} : Int;   // Length of the gap downstream (mm)
         GapToBeRecovered { ExternalAccessible := 'False'; ExternalVisible := 'False'; ExternalWritable := 'False'} : Int;   // Length of the recovered gap (mm)
         GapCovered { ExternalAccessible := 'False'; ExternalVisible := 'False'; ExternalWritable := 'False'} : Int;   // Length of  the covered gap (mm)
         LogNr { ExternalAccessible := 'False'; ExternalVisible := 'False'; ExternalWritable := 'False'} : Int;
         Accelerate { ExternalAccessible := 'False'; ExternalVisible := 'False'; ExternalWritable := 'False'} : Bool;   // True is acceleration needed
         Decelerate { ExternalAccessible := 'False'; ExternalVisible := 'False'; ExternalWritable := 'False'} : Bool;   // True is deceleration needed
      END_STRUCT;
      R_TRIG_PEC_Upstream {InstructionName := 'R_TRIG'; LibVersion := '1.0'; ExternalAccessible := 'False'; ExternalVisible := 'False'; ExternalWritable := 'False'; S7_SetPoint := 'False'} : R_TRIG;   // Rising triggering of the 2ste PEC of the upstream conveyor
      F_TRIG_PEC_Upstream {InstructionName := 'F_TRIG'; LibVersion := '1.0'; ExternalAccessible := 'False'; ExternalVisible := 'False'; ExternalWritable := 'False'; S7_SetPoint := 'False'} : F_TRIG;   // Falling triggering of the 2ste PEC of the upstream conveyor
      R_TRIG_PEC_Downstream {InstructionName := 'R_TRIG'; LibVersion := '1.0'; ExternalAccessible := 'False'; ExternalVisible := 'False'; ExternalWritable := 'False'; S7_SetPoint := 'False'} : R_TRIG;   // Rising triggering of the PEC of the downstream conveyor
      F_TRIG_PEC_Downstream {InstructionName := 'F_TRIG'; LibVersion := '1.0'; ExternalAccessible := 'False'; ExternalVisible := 'False'; ExternalWritable := 'False'; S7_SetPoint := 'False'} : F_TRIG;   // Falling triggering of the PEC of the downstream conveyor
      F_TRIG_PEC_A1 {InstructionName := 'F_TRIG'; LibVersion := '1.0'; ExternalAccessible := 'False'; ExternalVisible := 'False'; ExternalWritable := 'False'; S7_SetPoint := 'False'} : F_TRIG;   // Falling triggering of the 1ste PEC of conveyor A
      F_TRIG_PEC_A2 {InstructionName := 'F_TRIG'; LibVersion := '1.0'; ExternalAccessible := 'False'; ExternalVisible := 'False'; ExternalWritable := 'False'; S7_SetPoint := 'False'} : F_TRIG;   // Falling triggering of the 2nd PEC of conveyor A
      F_TRIG_PEC_B1 {InstructionName := 'F_TRIG'; LibVersion := '1.0'; ExternalAccessible := 'False'; ExternalVisible := 'False'; ExternalWritable := 'False'; S7_SetPoint := 'False'} : F_TRIG;   // Falling triggering of the 1ste PEC of conveyor B
      F_TRIG_PEC_B2 {InstructionName := 'F_TRIG'; LibVersion := '1.0'; ExternalAccessible := 'False'; ExternalVisible := 'False'; ExternalWritable := 'False'; S7_SetPoint := 'False'} : F_TRIG;   // Falling triggering of the 2nd PEC of conveyor B
      F_TRIG_PEC_C1 {InstructionName := 'F_TRIG'; LibVersion := '1.0'; ExternalAccessible := 'False'; ExternalVisible := 'False'; ExternalWritable := 'False'; S7_SetPoint := 'False'} : F_TRIG;   // Falling triggering of the 1ste PEC of conveyor C
      F_TRIG_PEC_C2 {InstructionName := 'F_TRIG'; LibVersion := '1.0'; ExternalAccessible := 'False'; ExternalVisible := 'False'; ExternalWritable := 'False'; S7_SetPoint := 'False'} : F_TRIG;   // Falling triggering of the 2nd PEC of conveyor C
      R_TRIG_PEC_A1 {InstructionName := 'R_TRIG'; LibVersion := '1.0'; ExternalAccessible := 'False'; ExternalVisible := 'False'; ExternalWritable := 'False'; S7_SetPoint := 'False'} : R_TRIG;   // Rising triggering of the 1ste PEC of conveyor A
      R_TRIG_PEC_A2 {InstructionName := 'R_TRIG'; LibVersion := '1.0'; ExternalAccessible := 'False'; ExternalVisible := 'False'; ExternalWritable := 'False'; S7_SetPoint := 'False'} : R_TRIG;   // Rising triggering of the 2nd PEC of conveyor A
      R_TRIG_PEC_B1 {InstructionName := 'R_TRIG'; LibVersion := '1.0'; ExternalAccessible := 'False'; ExternalVisible := 'False'; ExternalWritable := 'False'; S7_SetPoint := 'False'} : R_TRIG;   // Rising triggering of the 1ste PEC of conveyor B
      R_TRIG_PEC_B2 {InstructionName := 'R_TRIG'; LibVersion := '1.0'; ExternalAccessible := 'False'; ExternalVisible := 'False'; ExternalWritable := 'False'; S7_SetPoint := 'False'} : R_TRIG;   // Rising triggering of the 2nd PEC of conveyor B
      R_TRIG_PEC_C1 {InstructionName := 'R_TRIG'; LibVersion := '1.0'; ExternalAccessible := 'False'; ExternalVisible := 'False'; ExternalWritable := 'False'; S7_SetPoint := 'False'} : R_TRIG;   // Rising triggering of the 1ste PEC of conveyor C
      R_TRIG_PEC_C2 {InstructionName := 'R_TRIG'; LibVersion := '1.0'; ExternalAccessible := 'False'; ExternalVisible := 'False'; ExternalWritable := 'False'; S7_SetPoint := 'False'} : R_TRIG;   // Rising triggering of the 2nd PEC of conveyor C
      R_TRIG_DataStartConvA {InstructionName := 'R_TRIG'; LibVersion := '1.0'; ExternalAccessible := 'False'; ExternalVisible := 'False'; ExternalWritable := 'False'; S7_SetPoint := 'False'} : R_TRIG;
      R_TRIG_DataStartConvB {InstructionName := 'R_TRIG'; LibVersion := '1.0'; ExternalAccessible := 'False'; ExternalVisible := 'False'; ExternalWritable := 'False'; S7_SetPoint := 'False'} : R_TRIG;
      R_TRIG_DataStartConvC {InstructionName := 'R_TRIG'; LibVersion := '1.0'; ExternalAccessible := 'False'; ExternalVisible := 'False'; ExternalWritable := 'False'; S7_SetPoint := 'False'} : R_TRIG;
      F_TRIG_TwoParcelsOnConvA {InstructionName := 'F_TRIG'; LibVersion := '1.0'; ExternalAccessible := 'False'; ExternalVisible := 'False'; ExternalWritable := 'False'; S7_SetPoint := 'False'} : F_TRIG;
      F_TRIG_TwoParcelsOnConvB {InstructionName := 'F_TRIG'; LibVersion := '1.0'; ExternalAccessible := 'False'; ExternalVisible := 'False'; ExternalWritable := 'False'; S7_SetPoint := 'False'} : F_TRIG;
      F_TRIG_TwoParcelsOnConvC {InstructionName := 'F_TRIG'; LibVersion := '1.0'; ExternalAccessible := 'False'; ExternalVisible := 'False'; ExternalWritable := 'False'; S7_SetPoint := 'False'} : F_TRIG;
      Slr_TimeSpeedChangeConvA { ExternalAccessible := 'False'; ExternalVisible := 'False'; ExternalWritable := 'False'} : LReal;
      Slr_TimeSpeedChangeConvB { ExternalAccessible := 'False'; ExternalVisible := 'False'; ExternalWritable := 'False'} : LReal;
      Slr_TimeSpeedChangeConvC { ExternalAccessible := 'False'; ExternalVisible := 'False'; ExternalWritable := 'False'} : LReal;
      si_CountNr { ExternalAccessible := 'False'; ExternalVisible := 'False'; ExternalWritable := 'False'} : Int;   // Counting the amount of parcels
      si_SpeedA { ExternalAccessible := 'False'; ExternalVisible := 'False'; ExternalWritable := 'False'} : Int;   // Setpoint speed for conveyor A (mm/s)
      si_SpeedB { ExternalAccessible := 'False'; ExternalVisible := 'False'; ExternalWritable := 'False'} : Int;   // Setpoint speed for conveyor B (mm/s)
      si_SpeedC { ExternalAccessible := 'False'; ExternalVisible := 'False'; ExternalWritable := 'False'} : Int;   // Setpoint speed for conveyor C (mm/s)
      si_DistanceTravelled_A_B { ExternalAccessible := 'False'; ExternalVisible := 'False'; ExternalWritable := 'False'} : Int;   // Distance travelled for conveyor A and B (mm)
      si_DistanceTravelled_B_C { ExternalAccessible := 'False'; ExternalVisible := 'False'; ExternalWritable := 'False'} : Int;   // Distance travelled for conveyor B and C (mm)
      si_ParcelGapRecovered_A { ExternalAccessible := 'False'; ExternalVisible := 'False'; ExternalWritable := 'False'} : Int;   // Actual gap that is recovered by conveyor A
      si_ParcelGapRecovered_C { ExternalAccessible := 'False'; ExternalVisible := 'False'; ExternalWritable := 'False'} : Int;   // Actual gap that is recovered by conveyor B
      si_ParcelGapRecovered_B { ExternalAccessible := 'False'; ExternalVisible := 'False'; ExternalWritable := 'False'} : Int;   // Actual gap that is recovered by conveyor C
      si_ParcelDownStreamResults { ExternalAccessible := 'False'; ExternalVisible := 'False'; ExternalWritable := 'False'} : Int;   // The result of the downstream gap recovered
      si_LoopCounter { ExternalAccessible := 'False'; ExternalVisible := 'False'; ExternalWritable := 'False'} : Int;   // Counter for loop
      si_MaxNumberofEntries { ExternalAccessible := 'False'; ExternalVisible := 'False'; ExternalWritable := 'False'} : Int;   // Maximum number of FIFO entries
      si_ReturnValue { ExternalAccessible := 'False'; ExternalVisible := 'False'; ExternalWritable := 'False'} : Int;   // Info Code of Move Block Siemens
      s_ConveyorA_GIN1 { ExternalAccessible := 'False'; ExternalVisible := 'False'; ExternalWritable := 'False'} : Int;
      s_ConveyorA_GIN2 { ExternalAccessible := 'False'; ExternalVisible := 'False'; ExternalWritable := 'False'} : Int;
      s_ConveyorB_GIN1 { ExternalAccessible := 'False'; ExternalVisible := 'False'; ExternalWritable := 'False'} : Int;
      s_ConveyorB_GIN2 { ExternalAccessible := 'False'; ExternalVisible := 'False'; ExternalWritable := 'False'} : Int;
      s_ConveyorC_GIN1 { ExternalAccessible := 'False'; ExternalVisible := 'False'; ExternalWritable := 'False'} : Int;
      s_ConveyorC_GIN2 { ExternalAccessible := 'False'; ExternalVisible := 'False'; ExternalWritable := 'False'} : Int;
      s_TailPositionParcelA { ExternalAccessible := 'False'; ExternalVisible := 'False'; ExternalWritable := 'False'} : Int;
      s_TailPositionParcelB { ExternalAccessible := 'False'; ExternalVisible := 'False'; ExternalWritable := 'False'} : Int;
      s_TailPositionParcelC { ExternalAccessible := 'False'; ExternalVisible := 'False'; ExternalWritable := 'False'} : Int;
      sx_ParcelsOnConveyor_A { ExternalAccessible := 'False'; ExternalVisible := 'False'; ExternalWritable := 'False'} : Bool;   // True = parcel is on the conveyor A
      sx_ParcelsOnConveyor_B { ExternalAccessible := 'False'; ExternalVisible := 'False'; ExternalWritable := 'False'} : Bool := FALSE;   // True = parcel is on the conveyor B
      sx_ParcelsOnConveyor_C { ExternalAccessible := 'False'; ExternalVisible := 'False'; ExternalWritable := 'False'} : Bool := FALSE;   // True = parcel is on the conveyor C
      sx_ActionConv_A { ExternalAccessible := 'False'; ExternalVisible := 'False'; ExternalWritable := 'False'} : Bool;   // True = release for the conveyor to get the setpoint
      sx_ActionConv_B { ExternalAccessible := 'False'; ExternalVisible := 'False'; ExternalWritable := 'False'} : Bool;   // True = release for the conveyor to get the setpoint
      sx_ActionConv_C { ExternalAccessible := 'False'; ExternalVisible := 'False'; ExternalWritable := 'False'} : Bool;   // True = release for the conveyor to get the setpoint
      sx_WaitCurrentParcel_A_B { ExternalAccessible := 'False'; ExternalVisible := 'False'; ExternalWritable := 'False'} : Bool;   // True = wait till next parcel left the next conveyor and then calculate again
      sx_WaitCurrentParcel_B_C { ExternalAccessible := 'False'; ExternalVisible := 'False'; ExternalWritable := 'False'} : Bool;   // True = wait till next parcel left the next conveyor and then calculate again
      sx_anotherparcelonConveyorB { ExternalAccessible := 'False'; ExternalVisible := 'False'; ExternalWritable := 'False'} : Bool;
      sr_TravelDistance_CurrentnewParc_B { ExternalAccessible := 'False'; ExternalVisible := 'False'; ExternalWritable := 'False'} : Real;
      sx_twoParcelsOnConveyor_A { ExternalAccessible := 'False'; ExternalVisible := 'False'; ExternalWritable := 'False'} : Bool;
      sx_twoParcelsOnConveyor_B { ExternalAccessible := 'False'; ExternalVisible := 'False'; ExternalWritable := 'False'} : Bool;
      sx_twoParcelsOnConveyor_C { ExternalAccessible := 'False'; ExternalVisible := 'False'; ExternalWritable := 'False'} : Bool;
      SetNominalSpeedA { ExternalAccessible := 'False'; ExternalVisible := 'False'; ExternalWritable := 'False'} : Bool;
      SetNominalSpeedB { ExternalAccessible := 'False'; ExternalVisible := 'False'; ExternalWritable := 'False'} : Bool;
      SetNominalSpeedC { ExternalAccessible := 'False'; ExternalVisible := 'False'; ExternalWritable := 'False'} : Bool;
   END_VAR


BEGIN
	(*
	----------------------------------------------------------------------------------------

	Version history:
	Date        | Version   | Author        | Remark
	----------------------------------------------------------------------------------------
	21/01/2020  | 1.0       | R. Joosse     | first release TIA 15.1
	04/04/2023  | 4.0       | F.Baten       | 4.0 Release TIA 17.5
	12/02/2024  | 4.1       | S.Nieswiec    | Variable name changes according to standard
	*)
	REGION 1 - Initialize

	    REGION 1.1 Firstscan

	        IF "DB_Memory".FirstScan THEN
	            #si_SpeedA := #ii_LoopSpeed;
	            #si_SpeedB := #ii_LoopSpeed;
	            #si_SpeedC := #ii_LoopSpeed;
	        END_IF;
	        #s_ConveyorA_GIN1 := 0;
	        #s_ConveyorA_GIN2 := 0;
	        #s_TailPositionParcelA := 0;
	        #s_ConveyorB_GIN1 := 0;
	        #s_ConveyorB_GIN2 := 0;
	        #s_TailPositionParcelB := 0;
	        #s_ConveyorC_GIN1 := 0;
	        #s_ConveyorC_GIN2 := 0;
	        #s_TailPositionParcelC := 0;

	    END_REGION

	    REGION 1.2 Triggers

	        #R_TRIG_PEC_Upstream(CLK := #ix_PECUpstream);
	        #F_TRIG_PEC_Upstream(CLK := #ix_PECUpstream);
	        #F_TRIG_PEC_A1(CLK := #ix_PECA1);
	        #R_TRIG_PEC_A1(CLK := #ix_PECA1);
	        #F_TRIG_PEC_A2(CLK := #ix_PECA2);
	        #R_TRIG_PEC_A2(CLK := #ix_PECA2);
	        #F_TRIG_PEC_B1(CLK := #ix_PECB1);
	        #R_TRIG_PEC_B1(CLK := #ix_PECB1);
	        #F_TRIG_PEC_B2(CLK := #ix_PECB2);
	        #R_TRIG_PEC_B2(CLK := #ix_PECB2);
	        #F_TRIG_PEC_C1(CLK := #ix_PECC1);
	        #R_TRIG_PEC_C1(CLK := #ix_PECC1);
	        #F_TRIG_PEC_C2(CLK := #ix_PECC2);
	        #R_TRIG_PEC_C2(CLK := #ix_PECC2);
	        #R_TRIG_PEC_Downstream(CLK := #ix_PECDownstream);
	        #F_TRIG_PEC_Downstream(CLK := #ix_PECDownstream);
	        #R_TRIG_DataStartConvA(CLK := (#iqa_TrackingDataUpstream[10] = 0)); // [#i_UDT_GOSConfiguration.Length_Conv_A /10]) = 0 );
	        #R_TRIG_DataStartConvB(CLK := (#iqa_TrackingDataA[10]) = 0);
	        #R_TRIG_DataStartConvC(CLK := (#iqa_TrackingDataB[10]) = 0);


	    END_REGION
	END_REGION

	REGION 2- Startup

	    REGION 2.1 - Check parcels on the conveyors
	        //set or reset bit when parcel is on the conveyor or left the conveyor by checking the Tracking Array

	        FOR #si_LoopCounter := 15 TO 95 BY 5 DO

	            IF #iqa_TrackingDataA[#si_LoopCounter] > 0
	            THEN
	                #sx_ParcelsOnConveyor_A := TRUE;
	                EXIT;
	            ELSE
	                #sx_ParcelsOnConveyor_A := FALSE;
	            END_IF;
	        END_FOR;

	        FOR #si_LoopCounter := 15 TO 95 BY 5 DO

	            IF #iqa_TrackingDataB[#si_LoopCounter] > 0
	            THEN
	                #sx_ParcelsOnConveyor_B := TRUE;
	                EXIT;
	            ELSE
	                #sx_ParcelsOnConveyor_B := FALSE;
	            END_IF;
	        END_FOR;

	        FOR #si_LoopCounter := 15 TO 95 BY 5 DO

	            IF #iqa_TrackingDataC[#si_LoopCounter] > 0
	            THEN
	                #sx_ParcelsOnConveyor_C := TRUE;
	                EXIT;
	            ELSE
	                #sx_ParcelsOnConveyor_C := FALSE;
	            END_IF;
	        END_FOR;


	        FOR #si_LoopCounter := 95 TO 5 BY -1 DO

	            IF #iqa_TrackingDataA[#si_LoopCounter] > 0
	            THEN
	                IF #s_ConveyorA_GIN1 = 0
	                THEN
	                    #s_ConveyorA_GIN1 := #iqa_TrackingDataA[#si_LoopCounter];
	                    #sx_twoParcelsOnConveyor_A := FALSE;
	                    #s_TailPositionParcelA := ((#iUDT_GOSConfiguration.LengthConvA / 10) - #si_LoopCounter);
	                END_IF;
	                IF #iqa_TrackingDataA[#si_LoopCounter] <> #s_ConveyorA_GIN1 AND #iqa_TrackingDataA[#si_LoopCounter] > 0
	                THEN
	                    #s_ConveyorA_GIN2 := #iqa_TrackingDataA[#si_LoopCounter];
	                    #sx_twoParcelsOnConveyor_A := TRUE;
	                END_IF;
	                //  EXIT;
	            ELSE
	                #sx_twoParcelsOnConveyor_A := FALSE;
	            END_IF;
	        END_FOR;

	        #F_TRIG_TwoParcelsOnConvA(CLK := #sx_twoParcelsOnConveyor_A);

	        // COnveyor B
	        FOR #si_LoopCounter := 95 TO 5 BY -1 DO

	            IF #iqa_TrackingDataB[#si_LoopCounter] > 0
	            THEN
	                IF #s_ConveyorB_GIN1 = 0
	                THEN
	                    #s_ConveyorB_GIN1 := #iqa_TrackingDataB[#si_LoopCounter];
	                    #sx_twoParcelsOnConveyor_B := FALSE;
	                    #s_TailPositionParcelB := ((#iUDT_GOSConfiguration.LengthConvB / 10) - #si_LoopCounter);
	                END_IF;
	                IF #iqa_TrackingDataB[#si_LoopCounter] <> #s_ConveyorB_GIN1 AND #iqa_TrackingDataB[#si_LoopCounter] > 0
	                THEN
	                    #s_ConveyorB_GIN2 := #iqa_TrackingDataB[#si_LoopCounter];
	                    #sx_twoParcelsOnConveyor_B := TRUE;
	                END_IF;
	                //  EXIT;
	            ELSE
	                #sx_twoParcelsOnConveyor_B := FALSE;
	            END_IF;
	        END_FOR;

	        #F_TRIG_TwoParcelsOnConvB(CLK := #sx_twoParcelsOnConveyor_B);

	        // COnveyor C
	        FOR #si_LoopCounter := 95 TO 5 BY -1 DO

	            IF #iqa_TrackingDataC[#si_LoopCounter] > 0
	            THEN
	                IF #s_ConveyorC_GIN1 = 0
	                THEN
	                    #s_ConveyorC_GIN1 := #iqa_TrackingDataC[#si_LoopCounter];
	                    #sx_twoParcelsOnConveyor_C := FALSE;
	                    #s_TailPositionParcelC := ((#iUDT_GOSConfiguration.LengthConvC / 10) - #si_LoopCounter);
	                END_IF;
	                IF #iqa_TrackingDataC[#si_LoopCounter] <> #s_ConveyorC_GIN1 AND #iqa_TrackingDataC[#si_LoopCounter] > 0
	                THEN
	                    #s_ConveyorC_GIN2 := #iqa_TrackingDataC[#si_LoopCounter];
	                    #sx_twoParcelsOnConveyor_C := TRUE;
	                END_IF;
	                //  EXIT;
	            ELSE
	                #sx_twoParcelsOnConveyor_C := FALSE;
	            END_IF;
	        END_FOR;

	        #F_TRIG_TwoParcelsOnConvC(CLK := #sx_twoParcelsOnConveyor_C);
	    END_REGION

	    REGION 2.2 Take data from GIN record
	        IF #R_TRIG_DataStartConvA.Q // #R_TRIG_PEC_A1.Q
	        THEN
	            #sa_ParcelA1.GIN := (#iqa_TrackingDataUpstream[5]);
	            //  #ss_ParcelA1.GIN := #iqs_TrackingData_A[(#i_UDT_GOSConfiguration.Pos_PEC_A1 / 10) - 5];
	            #sa_ParcelA1.GapUpstream := 0;
	            #sa_ParcelA1.GapDownstream := 0;
	            IF #sa_ParcelA1.GIN > 0
	            THEN
	                #sa_ParcelA1.Length := ("DB_GIN".GIN[#sa_ParcelA1.GIN].General.Length * 10);
	                #sa_ParcelA1.GapUpstream := ("DB_GIN".GIN[#sa_ParcelA1.GIN].General.TrailingGap * 10);
	                #sa_ParcelA1.GapDownstream := ("DB_GIN".GIN[#sa_ParcelA1.GIN].General.LeadingGap * 10);

	                IF "DB_GIN".GIN[#sa_ParcelA1.GIN].General.LeadingGap > 3200
	                THEN
	                    #sa_ParcelA1.GapDownstream := 10000;
	                END_IF;

	                IF "DB_GIN".GIN[#sa_ParcelA1.GIN].General.TrailingGap > 3200
	                THEN
	                    #sa_ParcelA1.GapUpstream := 10000;
	                END_IF;

	                #sa_ParcelA1.GapToBeRecovered := #sa_ParcelA1.GapDownstream - #iUDT_GOSConfiguration.RequiredGap;
	            END_IF;
	        END_IF;

	        IF #R_TRIG_DataStartConvB.Q//#R_TRIG_PEC_B1.Q
	        THEN
	            #sa_ParcelB1.GIN := #iqa_TrackingDataA[7];
	            #sa_ParcelB1.GapUpstream := 0;
	            #sa_ParcelB1.GapDownstream := 0;

	            IF #sa_ParcelB1.GIN > 0
	            THEN
	                #sa_ParcelB1.Length := ("DB_GIN".GIN[#sa_ParcelB1.GIN].General.Length * 10);
	                #sa_ParcelB1.GapUpstream := ("DB_GIN".GIN[#sa_ParcelB1.GIN].General.TrailingGap * 10);
	                #sa_ParcelB1.GapDownstream := ("DB_GIN".GIN[#sa_ParcelB1.GIN].General.LeadingGap * 10);

	                IF "DB_GIN".GIN[#sa_ParcelB1.GIN].General.LeadingGap > 3200
	                THEN
	                    #sa_ParcelB1.GapDownstream := 10000;
	                END_IF;

	                IF "DB_GIN".GIN[#sa_ParcelB1.GIN].General.TrailingGap > 3200
	                THEN
	                    #sa_ParcelB1.GapUpstream := 10000;
	                END_IF;
	                #sa_ParcelB1.GapToBeRecovered := #sa_ParcelB1.GapDownstream - #iUDT_GOSConfiguration.RequiredGap;
	            END_IF;
	        END_IF;

	        IF #R_TRIG_DataStartConvC.Q///#R_TRIG_PEC_C1.Q
	        THEN
	            #sa_ParcelC1.GIN := #iqa_TrackingDataB[7];
	            #sa_ParcelC1.GapUpstream := 0;
	            #sa_ParcelC1.GapDownstream := 0;

	            IF #sa_ParcelC1.GIN > 0
	            THEN
	                #sa_ParcelC1.Length := ("DB_GIN".GIN[#sa_ParcelC1.GIN].General.Length * 10);
	                #sa_ParcelC1.GapUpstream := ("DB_GIN".GIN[#sa_ParcelC1.GIN].General.TrailingGap * 10);
	                #sa_ParcelC1.GapDownstream := ("DB_GIN".GIN[#sa_ParcelC1.GIN].General.LeadingGap * 10);

	                IF "DB_GIN".GIN[#sa_ParcelC1.GIN].General.LeadingGap > 3200
	                THEN
	                    #sa_ParcelC1.GapDownstream := 10000;
	                END_IF;

	                IF "DB_GIN".GIN[#sa_ParcelC1.GIN].General.TrailingGap > 3200
	                THEN
	                    #sa_ParcelC1.GapUpstream := 10000;
	                END_IF;
	                #sa_ParcelC1.GapToBeRecovered := #sa_ParcelB1.GapDownstream - #iUDT_GOSConfiguration.RequiredGap;
	            END_IF;
	        END_IF;




	    END_REGION

	    REGION 2.3 - Calculations

	        REGION 2.3.1 Mode 100

	            IF ((#R_TRIG_DataStartConvA.Q AND NOT #sx_twoParcelsOnConveyor_A)//#R_TRIG_PEC_A1.Q
	                OR (#F_TRIG_TwoParcelsOnConvA.Q AND #iqa_TrackingDataUpstream[10] = 0))
	                AND NOT #sx_ParcelsOnConveyor_B
	                AND NOT #sx_ParcelsOnConveyor_C
	                AND NOT #sx_ActionConv_A
	                AND NOT #sx_ActionConv_B
	                AND NOT #sx_ActionConv_C
	            THEN
	                IF #R_TRIG_DataStartConvA.Q THEN
	                    #sr_TravelDistanceUpstreamParc := INT_TO_REAL(#sa_ParcelA1.GapUpstream) - INT_TO_REAL(#iUDT_GOSConfiguration.LengthSpaceBetweenConv);
	                    #sr_TravelDistanceCurrentParcA := (INT_TO_REAL(#iUDT_GOSConfiguration.LengthConvA - #sa_ParcelA1.Length) + INT_TO_REAL(#iUDT_GOSConfiguration.LengthConvB) + INT_TO_REAL(#iUDT_GOSConfiguration.LengthConvC) - INT_TO_REAL(#iUDT_GOSConfiguration.PosPECC2));
	                    #sx_ActionConv_A := True;
	                    #sx_ActionConv_B := True;
	                    #sx_ActionConv_C := True;
	                END_IF;
	                IF #F_TRIG_TwoParcelsOnConvA.Q THEN
	                    #sr_TravelDistanceUpstreamParc := INT_TO_REAL(#sa_ParcelA1.GapUpstream) - INT_TO_REAL(#iUDT_GOSConfiguration.LengthSpaceBetweenConv) - #s_TailPositionParcelA;
	                    #sr_TravelDistanceCurrentParcA := (INT_TO_REAL(#iUDT_GOSConfiguration.LengthConvA - #sa_ParcelA1.Length - #s_TailPositionParcelA) + INT_TO_REAL(#iUDT_GOSConfiguration.LengthConvB) + INT_TO_REAL(#iUDT_GOSConfiguration.LengthConvC) - INT_TO_REAL(#iUDT_GOSConfiguration.PosPECC2));
	                    #sx_ActionConv_A := True;
	                    #sx_ActionConv_B := True;
	                    #sx_ActionConv_C := True;
	                END_IF;
	                "FC_GOSCalculation"(ir_TravelDistanceCurrentParc := #sr_TravelDistanceCurrentParcA,
	                                    ir_TravelDistanceUpstreamParc := #sr_TravelDistanceUpstreamParc,
	                                    ir_InitialSpeed := #ii_LoopSpeed,
	                                    ir_Acceleration := #iUDT_GOSConfiguration.Acceleration,
	                                    ir_MaxSpeed := #iUDT_GOSConfiguration.MaximumSpeed,
	                                    ir_MinSpeed := #iUDT_GOSConfiguration.MinimumSpeed,
	                                    ii_ParcelGapDownstream := #sa_ParcelA1.GapDownstream,
	                                    ii_ParcelGapUpstream := #sa_ParcelA1.GapUpstream,
	                                    ii_RequiredGap := #iUDT_GOSConfiguration.RequiredGap,
	                                    ii_MarginGap := #iUDT_GOSConfiguration.MarginLength,
	                                    ii_AllowedUpstreamGap := #iUDT_GOSConfiguration.AllowedUpstreamGap,
	                                    ix_ActionConv := #sx_ActionConv_A,
	                                    qx_Accelerate => #sa_ParcelA1.Accelerate,
	                                    qx_Decelerate => #sa_ParcelA1.Decelerate,
	                                    qi_Speed => #si_SpeedA,
	                                    qi_ParcelGapRecovered => #sa_ParcelA1.GapCovered,
	                                    qi_TimeToChangeSpeed => #Slr_TimeSpeedChangeConvA);

	                #Slr_TimeSpeedChangeConvB := #Slr_TimeSpeedChangeConvA;
	                #Slr_TimeSpeedChangeConvC := #Slr_TimeSpeedChangeConvA;
	                #si_SpeedB := #si_SpeedA;
	                #si_SpeedC := #si_SpeedA;
	                #si_ParcelDownStreamResults := #si_ParcelGapRecovered_A;

	            END_IF;
	        END_REGION

	        REGION 2.3.2 Mode 110 or 111 TRIGGER A1

	            IF ((#R_TRIG_DataStartConvA.Q AND NOT #sx_twoParcelsOnConveyor_A)  // #R_TRIG_PEC_A1.Q
	                OR (#F_TRIG_TwoParcelsOnConvA.Q AND #iqa_TrackingDataUpstream[10] = 0))
	                AND #sx_ParcelsOnConveyor_B
	                AND NOT #sx_ActionConv_A
	            THEN
	                IF #sa_ParcelA1.Length <= #iUDT_GOSConfiguration.AllowedParcelLength
	                THEN
	                    IF #R_TRIG_DataStartConvA.Q THEN
	                        #sr_TravelDistanceCurrentParcA := INT_TO_REAL(#iUDT_GOSConfiguration.LengthConvA - #iUDT_GOSConfiguration.PosPECA2 - #sa_ParcelA1.Length);
	                        #sr_TravelDistanceUpstreamParc := INT_TO_REAL(#sa_ParcelA1.GapUpstream) - INT_TO_REAL(#iUDT_GOSConfiguration.LengthSpaceBetweenConv);
	                        #sx_ActionConv_A := True;
	                    END_IF;
	                    IF #F_TRIG_TwoParcelsOnConvA.Q THEN
	                        #sr_TravelDistanceCurrentParcA := INT_TO_REAL(#iUDT_GOSConfiguration.LengthConvA - #iUDT_GOSConfiguration.PosPECA2 - #sa_ParcelA1.Length - #s_TailPositionParcelA);
	                        #sr_TravelDistanceUpstreamParc := INT_TO_REAL(#sa_ParcelA1.GapUpstream) - INT_TO_REAL(#iUDT_GOSConfiguration.LengthSpaceBetweenConv - #s_TailPositionParcelA);
	                        #sx_ActionConv_A := True;
	                    END_IF;
	                    "FC_GOSCalculation"(ir_TravelDistanceCurrentParc := #sr_TravelDistanceCurrentParcA,
	                                        ir_TravelDistanceUpstreamParc := #sr_TravelDistanceUpstreamParc,
	                                        ir_InitialSpeed := #ii_LoopSpeed,
	                                        ir_Acceleration := #iUDT_GOSConfiguration.Acceleration,
	                                        ir_MaxSpeed := #iUDT_GOSConfiguration.MaximumSpeed,
	                                        ir_MinSpeed := #iUDT_GOSConfiguration.MinimumSpeed,
	                                        ii_ParcelGapDownstream := #sa_ParcelA1.GapDownstream,
	                                        ii_ParcelGapUpstream := #sa_ParcelA1.GapUpstream,
	                                        ii_RequiredGap := #iUDT_GOSConfiguration.RequiredGap,
	                                        ii_MarginGap := #iUDT_GOSConfiguration.MarginLength,
	                                        ii_AllowedUpstreamGap := #iUDT_GOSConfiguration.AllowedUpstreamGap,
	                                        ix_ActionConv := #sx_ActionConv_A,
	                                        qx_Accelerate => #sa_ParcelA1.Accelerate,
	                                        qx_Decelerate => #sa_ParcelA1.Decelerate,
	                                        qi_Speed => #si_SpeedA,
	                                        qi_ParcelGapRecovered => #si_ParcelGapRecovered_A,
	                                        qi_TimeToChangeSpeed => #Slr_TimeSpeedChangeConvA);

	                    #si_ParcelDownStreamResults := #sa_ParcelA1.GapDownstream + #si_ParcelGapRecovered_A;

	                    IF #si_ParcelDownStreamResults > #iUDT_GOSConfiguration.RequiredGap
	                    THEN
	                        #si_ParcelDownStreamResults := #iUDT_GOSConfiguration.RequiredGap;
	                    ELSE
	                        #sx_WaitCurrentParcel_A_B := True;
	                    END_IF;
	                ELSE
	                    #sx_WaitCurrentParcel_A_B := True;
	                END_IF;
	            END_IF;

	            IF #sx_WaitCurrentParcel_A_B
	            THEN
	                #si_DistanceTravelled_A_B += (#iUDT_ConvA.Displacement * 10);
	            END_IF;

	            IF #R_TRIG_PEC_B2.Q
	                AND #sx_WaitCurrentParcel_A_B
	                AND NOT #sx_ActionConv_A
	                AND NOT #sx_ActionConv_B
	            THEN
	                #sr_TravelDistanceUpstreamParc := INT_TO_REAL((#sa_ParcelA1.GapUpstream - #si_DistanceTravelled_A_B)) - INT_TO_REAL(#iUDT_GOSConfiguration.LengthSpaceBetweenConv);
	                #sr_TravelDistanceCurrentParcA := (INT_TO_REAL(#iUDT_GOSConfiguration.LengthConvA) + INT_TO_REAL(#iUDT_GOSConfiguration.LengthConvB)) - (INT_TO_REAL(#iUDT_GOSConfiguration.PosPECB2) + INT_TO_REAL(#sa_ParcelA1.Length) + INT_TO_REAL(#si_DistanceTravelled_A_B));
	                #sx_WaitCurrentParcel_A_B := False;
	                #si_DistanceTravelled_A_B := 0;
	                #sx_ActionConv_A := True;
	                #sx_ActionConv_B := True;
	                "FC_GOSCalculation"(ir_TravelDistanceCurrentParc := #sr_TravelDistanceCurrentParcA,
	                                    ir_TravelDistanceUpstreamParc := #sr_TravelDistanceUpstreamParc,
	                                    ir_InitialSpeed := #ii_LoopSpeed,
	                                    ir_Acceleration := #iUDT_GOSConfiguration.Acceleration,
	                                    ir_MaxSpeed := #iUDT_GOSConfiguration.MaximumSpeed,
	                                    ir_MinSpeed := #iUDT_GOSConfiguration.MinimumSpeed,
	                                    ii_ParcelGapDownstream := #sa_ParcelA1.GapDownstream,
	                                    ii_ParcelGapUpstream := #sa_ParcelA1.GapUpstream,
	                                    ii_RequiredGap := #iUDT_GOSConfiguration.RequiredGap,
	                                    ii_MarginGap := #iUDT_GOSConfiguration.MarginLength,
	                                    ii_AllowedUpstreamGap := #iUDT_GOSConfiguration.AllowedUpstreamGap,
	                                    ix_ActionConv := #sx_ActionConv_A,
	                                    qx_Accelerate => #sa_ParcelA1.Accelerate,
	                                    qx_Decelerate => #sa_ParcelA1.Decelerate,
	                                    qi_Speed => #si_SpeedA,
	                                    qi_ParcelGapRecovered => #si_ParcelGapRecovered_A,
	                                    qi_TimeToChangeSpeed => #Slr_TimeSpeedChangeConvA);
	                #si_SpeedB := #si_SpeedA;
	                #Slr_TimeSpeedChangeConvB := #Slr_TimeSpeedChangeConvA;
	                #si_ParcelDownStreamResults := #si_ParcelGapRecovered_A;
	            END_IF;
	        END_REGION

	        REGION 2.3.3 Mode 101 TRIGGER A1

	            IF (#R_TRIG_DataStartConvA.Q AND NOT #sx_twoParcelsOnConveyor_A)
	                AND NOT #sx_ParcelsOnConveyor_B
	                AND #sx_ParcelsOnConveyor_C
	                AND NOT #sx_ActionConv_A
	                AND NOT #sx_ActionConv_B
	            THEN
	                #sr_TravelDistanceCurrentParcA := INT_TO_REAL(#iUDT_GOSConfiguration.LengthConvA) - INT_TO_REAL(#iUDT_GOSConfiguration.PosPECA2) - INT_TO_REAL(#sa_ParcelA1.Length) + INT_TO_REAL(#iUDT_GOSConfiguration.LengthConvB);
	                #sr_TravelDistanceUpstreamParc := INT_TO_REAL(#sa_ParcelA1.GapUpstream) - INT_TO_REAL(#iUDT_GOSConfiguration.LengthSpaceBetweenConv);

	                #sx_ActionConv_A := True;
	                #sx_ActionConv_B := True;
	                "FC_GOSCalculation"(ir_TravelDistanceCurrentParc := #sr_TravelDistanceCurrentParcA,
	                                    ir_TravelDistanceUpstreamParc := #sr_TravelDistanceUpstreamParc,
	                                    ir_InitialSpeed := #ii_LoopSpeed,
	                                    ir_Acceleration := #iUDT_GOSConfiguration.Acceleration,
	                                    ir_MaxSpeed := #iUDT_GOSConfiguration.MaximumSpeed,
	                                    ir_MinSpeed := #iUDT_GOSConfiguration.MinimumSpeed,
	                                    ii_ParcelGapDownstream := #sa_ParcelA1.GapDownstream,
	                                    ii_ParcelGapUpstream := #sa_ParcelA1.GapUpstream,
	                                    ii_RequiredGap := #iUDT_GOSConfiguration.RequiredGap,
	                                    ii_MarginGap := #iUDT_GOSConfiguration.MarginLength,
	                                    ii_AllowedUpstreamGap := #iUDT_GOSConfiguration.AllowedUpstreamGap,
	                                    ix_ActionConv := #sx_ActionConv_A,
	                                    qx_Accelerate => #sa_ParcelA1.Accelerate,
	                                    qx_Decelerate => #sa_ParcelA1.Decelerate,
	                                    qi_Speed => #si_SpeedA,
	                                    qi_ParcelGapRecovered => #si_ParcelGapRecovered_A,
	                                    qi_TimeToChangeSpeed => #Slr_TimeSpeedChangeConvA);

	                #si_SpeedB := #si_SpeedA;
	                #Slr_TimeSpeedChangeConvB := #Slr_TimeSpeedChangeConvA;
	                #si_ParcelDownStreamResults := #si_ParcelGapRecovered_A * 2;
	            END_IF;
	        END_REGION

	        REGION 2.3.4 Mode 110 OR Mode 010 by TRIGGER B1

	            IF ((#R_TRIG_DataStartConvB.Q AND NOT #sx_twoParcelsOnConveyor_B)
	                OR (#F_TRIG_TwoParcelsOnConvB.Q AND #iqa_TrackingDataA[10] = 0))
	                AND NOT #sx_ParcelsOnConveyor_C
	                AND NOT #sx_ActionConv_B
	            THEN
	                IF #R_TRIG_DataStartConvB.Q THEN
	                    #sr_TravelDistanceCurrentParcB := INT_TO_REAL(#iUDT_GOSConfiguration.LengthConvB - #sa_ParcelB1.Length + #iUDT_GOSConfiguration.LengthConvC - #iUDT_GOSConfiguration.PosPECC2);
	                    #sr_TravelDistanceUpstreamParcA := INT_TO_REAL(#sa_ParcelB1.GapUpstream) - INT_TO_REAL(#iUDT_GOSConfiguration.LengthSpaceBetweenConv);
	                    #sx_ActionConv_B := True;
	                    #sx_ActionConv_C := True;
	                END_IF;
	                IF #F_TRIG_TwoParcelsOnConvB.Q THEN
	                    #sr_TravelDistanceCurrentParcB := INT_TO_REAL(#iUDT_GOSConfiguration.LengthConvB - #sa_ParcelB1.Length - #s_TailPositionParcelB + #iUDT_GOSConfiguration.LengthConvC - #iUDT_GOSConfiguration.PosPECC2);
	                    #sr_TravelDistanceUpstreamParcA := INT_TO_REAL(#sa_ParcelB1.GapUpstream - #s_TailPositionParcelB) - INT_TO_REAL(#iUDT_GOSConfiguration.LengthSpaceBetweenConv);
	                    #sx_ActionConv_B := True;
	                    #sx_ActionConv_C := True;
	                END_IF;
	                "FC_GOSCalculation"(ir_TravelDistanceCurrentParc := #sr_TravelDistanceCurrentParcB,
	                                    ir_TravelDistanceUpstreamParc := #sr_TravelDistanceUpstreamParcA,
	                                    ir_InitialSpeed := #ii_LoopSpeed,
	                                    ir_Acceleration := #iUDT_GOSConfiguration.Acceleration,
	                                    ir_MaxSpeed := #iUDT_GOSConfiguration.MaximumSpeed,
	                                    ir_MinSpeed := #iUDT_GOSConfiguration.MinimumSpeed,
	                                    ii_ParcelGapDownstream := #sa_ParcelB1.GapDownstream,
	                                    ii_ParcelGapUpstream := #sa_ParcelB1.GapUpstream,
	                                    ii_RequiredGap := #iUDT_GOSConfiguration.RequiredGap,
	                                    ii_MarginGap := #iUDT_GOSConfiguration.MarginLength,
	                                    ii_AllowedUpstreamGap := #iUDT_GOSConfiguration.AllowedUpstreamGap,
	                                    ix_ActionConv := #sx_ActionConv_B,
	                                    qx_Accelerate => #sa_ParcelB1.Accelerate,
	                                    qx_Decelerate => #sa_ParcelB1.Decelerate,
	                                    qi_Speed => #si_SpeedB,
	                                    qi_ParcelGapRecovered => #si_ParcelGapRecovered_B,
	                                    qi_TimeToChangeSpeed => #Slr_TimeSpeedChangeConvB);

	                #si_SpeedC := #si_SpeedB;
	                #Slr_TimeSpeedChangeConvC := #Slr_TimeSpeedChangeConvB;

	            END_IF;
	        END_REGION

	        REGION 2.3.5 Mode 011 by TRIGGER B1

	            IF ((#R_TRIG_DataStartConvB.Q AND NOT #sx_twoParcelsOnConveyor_B)
	                OR (#F_TRIG_TwoParcelsOnConvB.Q AND #iqa_TrackingDataA[10] = 0))
	                AND #sx_ParcelsOnConveyor_C
	                AND NOT #sx_ActionConv_B
	            THEN
	                IF #sa_ParcelB1.Length <= #iUDT_GOSConfiguration.AllowedParcelLength
	                THEN
	                    IF NOT #sx_ParcelsOnConveyor_A AND #sa_ParcelB1.GapUpstream = 0 THEN
	                        #sr_TravelDistanceUpstreamParcA := INT_TO_REAL(#iUDT_GOSConfiguration.LengthConvB + #sa_ParcelB1.GapUpstream) - INT_TO_REAL(#iUDT_GOSConfiguration.LengthSpaceBetweenConv);
	                    ELSE
	                        #sr_TravelDistanceUpstreamParcA := INT_TO_REAL(#sa_ParcelB1.GapUpstream) - #s_TailPositionParcelB - INT_TO_REAL(#iUDT_GOSConfiguration.LengthSpaceBetweenConv);
	                    END_IF;
	                    #sr_TravelDistanceCurrentParcB := INT_TO_REAL(#iUDT_GOSConfiguration.LengthConvB) - INT_TO_REAL(#sa_ParcelB1.Length) - #s_TailPositionParcelB;
	                    #s_ConveyorA_GIN2 := 0;
	                    #s_TailPositionParcelB := 0;
	                    ;
	                    #sx_ActionConv_B := True;
	                    "FC_GOSCalculation"(ir_TravelDistanceCurrentParc := #sr_TravelDistanceCurrentParcB,
	                                        ir_TravelDistanceUpstreamParc := #sr_TravelDistanceUpstreamParcA,
	                                        ir_InitialSpeed := #ii_LoopSpeed,
	                                        ir_Acceleration := #iUDT_GOSConfiguration.Acceleration,
	                                        ir_MaxSpeed := #iUDT_GOSConfiguration.MaximumSpeed,
	                                        ir_MinSpeed := #iUDT_GOSConfiguration.MinimumSpeed,
	                                        ii_ParcelGapDownstream := #sa_ParcelB1.GapDownstream,
	                                        ii_ParcelGapUpstream := #sa_ParcelB1.GapUpstream,
	                                        ii_RequiredGap := #iUDT_GOSConfiguration.RequiredGap,
	                                        ii_MarginGap := #iUDT_GOSConfiguration.MarginLength,
	                                        ii_AllowedUpstreamGap := #iUDT_GOSConfiguration.AllowedUpstreamGap,
	                                        ix_ActionConv := #sx_ActionConv_B,
	                                        qx_Accelerate => #sa_ParcelB1.Accelerate,
	                                        qx_Decelerate => #sa_ParcelB1.Decelerate,
	                                        qi_Speed => #si_SpeedB,
	                                        qi_ParcelGapRecovered => #si_ParcelGapRecovered_B,
	                                        qi_TimeToChangeSpeed => #Slr_TimeSpeedChangeConvB);

	                    #si_ParcelDownStreamResults := #sa_ParcelB1.GapDownstream + #si_ParcelGapRecovered_B;

	                    IF #si_ParcelDownStreamResults > #iUDT_GOSConfiguration.RequiredGap
	                    THEN
	                        #si_ParcelDownStreamResults := #iUDT_GOSConfiguration.RequiredGap;
	                    ELSE
	                        #sx_WaitCurrentParcel_B_C := True;
	                    END_IF;
	                ELSE
	                    #sx_WaitCurrentParcel_B_C := TRUE;
	                END_IF;
	            END_IF;

	            IF #sx_WaitCurrentParcel_B_C
	            THEN
	                #si_DistanceTravelled_B_C += (#iUDT_ConvB.Displacement * 10);
	            END_IF;
	        END_REGION

	        REGION 2.3.6 Mode 001 by TRIGGER C1

	            IF ((#R_TRIG_DataStartConvC.Q AND NOT #sx_twoParcelsOnConveyor_C)// #R_TRIG_PEC_C1.Q
	                OR (#F_TRIG_TwoParcelsOnConvC.Q AND #iqa_TrackingDataA[10] = 0))
	                AND NOT #sx_ActionConv_C

	            THEN
	                IF NOT #sx_ParcelsOnConveyor_A AND NOT #sx_ParcelsOnConveyor_B AND #sa_ParcelC1.GapUpstream = 0 THEN
	                    #sr_TravelDistanceUpstreamParcB := INT_TO_REAL(#iUDT_GOSConfiguration.LengthConvA + #iUDT_GOSConfiguration.LengthConvB + #sa_ParcelC1.GapUpstream) - INT_TO_REAL(#iUDT_GOSConfiguration.LengthSpaceBetweenConv);
	                ELSIF NOT #sx_ParcelsOnConveyor_B AND #sa_ParcelC1.GapUpstream = 0 THEN
	                    #sr_TravelDistanceUpstreamParcB := INT_TO_REAL(#iUDT_GOSConfiguration.LengthConvB + #sa_ParcelC1.GapUpstream) - INT_TO_REAL(#iUDT_GOSConfiguration.LengthSpaceBetweenConv);
	                ELSE
	                    #sr_TravelDistanceUpstreamParcB := INT_TO_REAL(#sa_ParcelC1.GapUpstream) - #s_TailPositionParcelC - INT_TO_REAL(#iUDT_GOSConfiguration.LengthSpaceBetweenConv);
	                END_IF;

	                #sr_TravelDistanceCurrentParcC := INT_TO_REAL(#iUDT_GOSConfiguration.LengthConvC - #iUDT_GOSConfiguration.PosPECC2 - #sa_ParcelC1.Length);
	                #sx_ActionConv_C := True;
	                "FC_GOSCalculation"(ir_TravelDistanceCurrentParc := #sr_TravelDistanceCurrentParcC,
	                                    ir_TravelDistanceUpstreamParc := #sr_TravelDistanceUpstreamParcB,
	                                    ir_InitialSpeed := #ii_LoopSpeed,
	                                    ir_Acceleration := #iUDT_GOSConfiguration.Acceleration,
	                                    ir_MaxSpeed := #iUDT_GOSConfiguration.MaximumSpeed,
	                                    ir_MinSpeed := #iUDT_GOSConfiguration.MinimumSpeed,
	                                    ii_ParcelGapDownstream := #sa_ParcelC1.GapDownstream,
	                                    ii_ParcelGapUpstream := #sa_ParcelC1.GapUpstream,
	                                    ii_RequiredGap := #iUDT_GOSConfiguration.RequiredGap,
	                                    ii_MarginGap := #iUDT_GOSConfiguration.MarginLength,
	                                    ii_AllowedUpstreamGap := #iUDT_GOSConfiguration.AllowedUpstreamGap,
	                                    ix_ActionConv := #sx_ActionConv_C,
	                                    qx_Accelerate => #sa_ParcelC1.Accelerate,
	                                    qx_Decelerate => #sa_ParcelC1.Decelerate,
	                                    qi_Speed => #si_SpeedC,
	                                    qi_ParcelGapRecovered => #si_ParcelGapRecovered_C,
	                                    qi_TimeToChangeSpeed => #Slr_TimeSpeedChangeConvC);

	            END_IF;
	        END_REGION
	    END_REGION
	END_REGION

	REGION 3 - Write setpoint speed
	    //When new actual speed is equals to the new setpoint then write the initial speed as the new setpoint

	    IF #Slr_TimeSpeedChangeConvA > 0.0 THEN

	        #Slr_TimeSpeedChangeConvA := #Slr_TimeSpeedChangeConvA - "DB_Memory".PrevCycleTime;
	        #SetNominalSpeedA := true;
	    ELSE
	        #Slr_TimeSpeedChangeConvA := 0;
	        #SetNominalSpeedA := FALSE;
	    END_IF;

	    IF #Slr_TimeSpeedChangeConvB > 0.0 THEN

	        #Slr_TimeSpeedChangeConvB := #Slr_TimeSpeedChangeConvB - "DB_Memory".PrevCycleTime;
	        #SetNominalSpeedB := true;
	    ELSE
	        #Slr_TimeSpeedChangeConvB := 0;
	        #SetNominalSpeedB := FALSE;
	    END_IF;

	    IF #Slr_TimeSpeedChangeConvC > 0.0 THEN

	        #Slr_TimeSpeedChangeConvC := #Slr_TimeSpeedChangeConvC - "DB_Memory".PrevCycleTime;
	        #SetNominalSpeedC := true;
	    ELSE
	        #Slr_TimeSpeedChangeConvC := 0;
	        #SetNominalSpeedC := FALSE;
	    END_IF;


	    IF (#sx_ActionConv_A AND #SetNominalSpeedA AND #si_SpeedA > #ii_LoopSpeed)

	    THEN
	        #si_SpeedA := #iUDT_GOSConfiguration.MaximumSpeed;
	    ELSIF (#sx_ActionConv_A AND #SetNominalSpeedA AND #si_SpeedA < #ii_LoopSpeed)
	    THEN
	        #si_SpeedA := #iUDT_GOSConfiguration.MinimumSpeed;
	    END_IF;

	    IF (#sx_ActionConv_A AND #Slr_TimeSpeedChangeConvA <= 0)
	    THEN
	        #si_SpeedA := #ii_LoopSpeed;
	        #sx_ActionConv_A := FALSE;
	        #SetNominalSpeedA := FALSE;
	    END_IF;

	    IF (#sx_ActionConv_B AND #SetNominalSpeedB AND #si_SpeedB > #ii_LoopSpeed)
	    THEN
	        #si_SpeedB := #iUDT_GOSConfiguration.MaximumSpeed;
	    ELSIF (#sx_ActionConv_B AND #SetNominalSpeedB AND #si_SpeedB < #ii_LoopSpeed)
	    THEN
	        #si_SpeedB := #iUDT_GOSConfiguration.MinimumSpeed;
	    END_IF;

	    IF (#sx_ActionConv_B AND #Slr_TimeSpeedChangeConvB <= 0)
	    THEN
	        #si_SpeedB := #ii_LoopSpeed;
	        #sx_ActionConv_B := FALSE;
	        #SetNominalSpeedB := FALSE;
	    END_IF;

	    IF (#sx_ActionConv_C AND #SetNominalSpeedC AND #si_SpeedC > #ii_LoopSpeed)
	    THEN
	        #si_SpeedC := #iUDT_GOSConfiguration.MaximumSpeed;
	    ELSIF (#sx_ActionConv_C AND #SetNominalSpeedC AND #si_SpeedC < #ii_LoopSpeed)
	    THEN
	        #si_SpeedC := #iUDT_GOSConfiguration.MinimumSpeed;
	    END_IF;

	    IF (#sx_ActionConv_C AND #Slr_TimeSpeedChangeConvC <= 0)
	    THEN
	        #si_SpeedC := #ii_LoopSpeed;
	        #sx_ActionConv_C := FALSE;
	        #SetNominalSpeedC := FALSE;
	    END_IF;

	    //Write new setpoint speed in the UDT_GOSInterface
	    #iqUDT_GOSInterface.SpeedConvA := #si_SpeedA;
	    #iqUDT_GOSInterface.SpeedConvB := #si_SpeedB;
	    #iqUDT_GOSInterface.SpeedConvC := #si_SpeedC;

	END_REGION

	REGION 4 Logging

	    //Get size of FIFO array (without the zero)
	    #si_MaxNumberofEntries := ("FC_GetNrOfArrayEl"(#iqUDT_GOSLog) - 1);

	    //Write DB_GOSLog with the parcel values
	    IF (#R_TRIG_PEC_A1.Q AND NOT #sx_twoParcelsOnConveyor_A)
	        OR #F_TRIG_TwoParcelsOnConvA.Q
	        AND #sa_ParcelA1.GIN > 0
	    THEN

	        FOR #si_LoopCounter := 1 TO #si_MaxNumberofEntries DO
	            IF "DB_GOSLog".DB_GOSLog[#si_LoopCounter].GIN_nr = #sa_ParcelA1.GIN THEN

	                "DB_GOSLog".DB_GOSLog[#si_LoopCounter].GIN_nr := #sa_ParcelA1.GIN;
	                "DB_GOSLog".DB_GOSLog[#si_LoopCounter].ParcelLength := #sa_ParcelA1.Length;
	                "DB_GOSLog".DB_GOSLog[#si_LoopCounter].InfeedUpstreamGap := #sa_ParcelA1.GapUpstream;
	                "DB_GOSLog".DB_GOSLog[#si_LoopCounter].InfeedDownstreamGap := #sa_ParcelA1.GapDownstream;
	                "DB_GOSLog".DB_GOSLog[#si_LoopCounter].Accelerate := #sa_ParcelA1.Accelerate;
	                "DB_GOSLog".DB_GOSLog[#si_LoopCounter].Decelerate := #sa_ParcelA1.Decelerate;
	                "DB_GOSLog".DB_GOSLog[#si_LoopCounter].GapToBeRecovered := #sa_ParcelA1.GapToBeRecovered;

	                EXIT;
	            END_IF;
	        END_FOR;
	    END_IF;


	    IF #R_TRIG_PEC_C2.Q
	    THEN
	        #sa_ParcelC2.GIN := #iqa_TrackingDataC[(#iUDT_GOSConfiguration.PosPECC2 / 10) - 5];
	        IF #sa_ParcelC2.GIN > 0
	        THEN
	            FOR #si_LoopCounter := 1 TO #si_MaxNumberofEntries DO
	                IF "DB_GOSLog".DB_GOSLog[#si_LoopCounter].GIN_nr = #sa_ParcelC2.GIN THEN
	                    "DB_GOSLog".DB_GOSLog[#si_LoopCounter].OutfeedDownstreamGap := "DB_GIN".GIN[#sa_ParcelC2.GIN].General.LeadingGap * 10;
	                    "DB_GOSLog".DB_GOSLog[#si_LoopCounter].OutfeedUpstreamGap := "DB_GIN".GIN[#sa_ParcelC2.GIN].General.TrailingGap * 10;
	                    "DB_GOSLog".DB_GOSLog[#si_LoopCounter].ParcelDownStreamResults := #si_ParcelDownStreamResults; // this should be here
	                    EXIT;
	                END_IF;
	            END_FOR;
	        END_IF;

	    END_IF;

	END_REGION

	REGION 2 - Update/shift FIFO


	    // Handle shift request merge (FIFO entry is handled induct code is generated in tracking DB)
	    IF #iqx_ShiftRequest
	    THEN
	        #si_ReturnValue := MOVE_BLK_VARIANT(SRC := #iqUDT_GOSLog,
	                                            COUNT := INT_TO_UDINT(#si_MaxNumberofEntries - 2),
	                                            SRC_INDEX := 0,
	                                            DEST_INDEX := 1,
	                                            DEST => #iqUDT_GOSLog);
	        //Reset values of 0 entry(used oly for shifting)
	        "DB_GOSLog".DB_GOSLog[0].GIN_nr := 0;
	        "DB_GOSLog".DB_GOSLog[0].ParcelLength := 0;
	        "DB_GOSLog".DB_GOSLog[0].InfeedUpstreamGap := 0;
	        "DB_GOSLog".DB_GOSLog[0].InfeedDownstreamGap := 0;
	        "DB_GOSLog".DB_GOSLog[0].Accelerate := 0;
	        "DB_GOSLog".DB_GOSLog[0].Decelerate := 0;
	        "DB_GOSLog".DB_GOSLog[0].GapToBeRecovered := 0;
	        "DB_GOSLog".DB_GOSLog[0].ParcelDownStreamResults := 0;
	        "DB_GOSLog".DB_GOSLog[0].OutfeedDownstreamGap := 0;
	        "DB_GOSLog".DB_GOSLog[0].OutfeedUpstreamGap := 0;
	        "DB_GOSLog".DB_GOSLog[0].ParcelUpStreamResults := 0;
	        "DB_GOSLog".DB_GOSLog[0].PrevConveyorDownstreamGap := 0;
	        "DB_GOSLog".DB_GOSLog[0].PrevConveyorUpstreamGap := 0;
	        "DB_GOSLog".DB_GOSLog[0].NextConveyorDownstreamGap := 0;
	        "DB_GOSLog".DB_GOSLog[0].NextConveyorUpstreamGap := 0;
	        // reset shift request
	        #iqx_ShiftRequest := False;

	    END_IF;
	END_REGION



END_FUNCTION_BLOCK

FUNCTION_BLOCK "FB_AMBASpiralVeyor"
{ S7_Optimized_Access := 'TRUE' }
VERSION : 0.1
// ATTRIBUTES
// AUTO_NUMBER = True
// BLOCK_NUMBER = 255
// END_ATTRIBUTES
   VAR_INPUT
      ix_HardwareOK { ExternalAccessible := 'False'; ExternalVisible := 'False'; ExternalWritable := 'False'} : Bool;   // TRUE when hardware is ok
      iudi_DelayHardwareOK { ExternalAccessible := 'False'; ExternalVisible := 'False'; ExternalWritable := 'False'} : UDInt;   // [ms] Delay time for hardware ok signal
      ix_ProxSwitchDriveShaft { ExternalAccessible := 'False'; ExternalVisible := 'False'; ExternalWritable := 'False'} : Bool;   // Proximity switch signal drive shaft detection
      ix_ProxSwitchIdlerShaft { ExternalAccessible := 'False'; ExternalVisible := 'False'; ExternalWritable := 'False'} : Bool;   // Proximity switch signal idler shaft detection
      ix_ProxSwitchSlat { ExternalAccessible := 'False'; ExternalVisible := 'False'; ExternalWritable := 'False'} : Bool;   // Proximity switch signal slat detection
   END_VAR

   VAR_IN_OUT
      iqUDT_Statistics : "UDT_SpiralVeyorStatistics";
      iqUDT_Status : "UDT_SpiralVeyorStatus";
      iqUDT_EquipmentControl : "UDT_EquipmentControl";
      iqUDT_CommonStatus : "UDT_CommonStatus";
   END_VAR

   VAR
      sFB_HardwareOK { ExternalAccessible := 'False'; ExternalVisible := 'False'; ExternalWritable := 'False'; S7_SetPoint := 'False'} : "FB_TimerOnOffDelay";   // Timer on/off delay for hardware ok signal
      sFB_SlatCheck { ExternalAccessible := 'False'; ExternalVisible := 'False'; ExternalWritable := 'False'; S7_SetPoint := 'False'} : "FB_AMBASpiralSlatCheck";
      sFB_ChainCheck { ExternalAccessible := 'False'; ExternalVisible := 'False'; ExternalWritable := 'False'; S7_SetPoint := 'False'} : "FB_AMBASpiralChainCheck";
   END_VAR


BEGIN
	(*
	Version history:
	Date        | Version   | Author              | Remark
	----------------------------------------------------------------------------------------
	 14/03/2022 | 1.0       | G.Vlooswijk         | Initial version for FedEx Milano
	 11/05/2022 | 2.0       | G.Vlooswijk         | Splitted inner and outerlane status
	 22/09/2022 | 2.1       | G.Vlooswijk         | Removed HMIStatus
	 03/06/2024 | 2.2       | J.Majer             | Adapted to current library
	*)

	REGION Input preparation

	    // Hardware ok timer
	    #sFB_HardwareOK(iudi_OnDelayTime := #iudi_DelayHardwareOK,
	                    ix_SignalToDelay := #ix_HardwareOK);

	END_REGION

	REGION Missing slat dection

	    #sFB_SlatCheck(ix_SlatDetection := #ix_ProxSwitchSlat,
	                   ix_HardwareOk := #sFB_HardwareOK.qx_DelayedSignal,
	                   iqx_MissingSlatDetected := #iqUDT_Status.MissingSlat,
	                   iqUDT_Statistics := #iqUDT_Statistics.MissingSlat,
	                   iqUDT_EquipmentControl := #iqUDT_EquipmentControl);

	END_REGION

	REGION Chain check

	    #sFB_ChainCheck(ix_ProxSwitchDriveShaft := #ix_ProxSwitchDriveShaft,
	                    ix_ProxSwitchIdlerShaft := #ix_ProxSwitchIdlerShaft,
	                    ix_HardwareOK := #sFB_HardwareOK.qx_DelayedSignal,
	                    iqx_BrokenChainDetected := #iqUDT_Status.BrokenChain,
	                    iqx_ChainOverlengthDetected := #iqUDT_Status.ChainOverlength,
	                    iqUDT_BrokenChainStatistics := #iqUDT_Statistics.BrokenChain,
	                    iqUDT_ChainOverlengthStatistics := #iqUDT_Statistics.ChainOverlength,
	                    iqUDT_EquipmentControl := #iqUDT_EquipmentControl);

	END_REGION

	REGION Update common status

	    //Set/reset warning state on spiralveyor warnings
	    IF #iqUDT_Status.ChainOverlength AND NOT #iqUDT_CommonStatus.Warning THEN
	        #iqUDT_CommonStatus.Warning := TRUE;
	    ELSIF NOT #iqUDT_Status.ChainOverlength AND #iqUDT_CommonStatus.Warning THEN
	        #iqUDT_CommonStatus.Warning := FALSE;
	    END_IF;

	    //Set/reset error status on spiralveyor faults
	    IF (#iqUDT_Status.BrokenChain OR #iqUDT_Status.MissingSlat) AND NOT #iqUDT_CommonStatus.Error THEN
	        #iqUDT_CommonStatus.Error := TRUE;
	    ELSIF NOT #iqUDT_Status.BrokenChain AND NOT #iqUDT_Status.MissingSlat AND #iqUDT_CommonStatus.Error THEN
	        #iqUDT_CommonStatus.Error := FALSE;
	    END_IF;

	END_REGION


END_FUNCTION_BLOCK

FUNCTION_BLOCK "FB_ControlPowerGroup"
TITLE = Control Power Group
{ S7_Optimized_Access := 'TRUE' }
AUTHOR : CesarLeite
VERSION : 3.0
// ATTRIBUTES
// AUTO_NUMBER = True
// BLOCK_NUMBER = 4
// END_ATTRIBUTES
//This block is used to monitoring the 24V power supplies.
   VAR_INPUT
      ix_PowerSupplyOk_1 { ExternalAccessible := 'False'; ExternalVisible := 'False'; ExternalWritable := 'False'} : Bool;   //  TRUE if power supply 1 is OK
      ix_PowerSupply_Infeed_1 { ExternalAccessible := 'False'; ExternalVisible := 'False'; ExternalWritable := 'False'} : Bool;   //  400V power supply 1 infeed
      ix_PowerSupplyOk_2 { ExternalAccessible := 'False'; ExternalVisible := 'False'; ExternalWritable := 'False'} : Bool;   //  TRUE if power supply 2 is OK
      ix_PowerSupply_Infeed_2 { ExternalAccessible := 'False'; ExternalVisible := 'False'; ExternalWritable := 'False'} : Bool;   //  400V power supply 2 infeed
      ix_PowerSupplyOk_3 { ExternalAccessible := 'False'; ExternalVisible := 'False'; ExternalWritable := 'False'} : Bool;   //  TRUE if power supply 3 is OK
      ix_PowerSupply_Infeed_3 { ExternalAccessible := 'False'; ExternalVisible := 'False'; ExternalWritable := 'False'} : Bool;   //  400V power supply 3 infeed
      ix_PowerSupplyOk_4 { ExternalAccessible := 'False'; ExternalVisible := 'False'; ExternalWritable := 'False'} : Bool;   //  TRUE if power supply 4 is OK
      ix_PowerSupply_Infeed_4 { ExternalAccessible := 'False'; ExternalVisible := 'False'; ExternalWritable := 'False'} : Bool;   //  400V power supply 4 infeed
      ix_PowerSupplyOk_5 { ExternalAccessible := 'False'; ExternalVisible := 'False'; ExternalWritable := 'False'} : Bool;   //  TRUE if power supply 5 is OK
      ix_PowerSupply_Infeed_5 { ExternalAccessible := 'False'; ExternalVisible := 'False'; ExternalWritable := 'False'} : Bool;   //  400V power supply 5 infeed
      ix_PowerSupplyOk_6 { ExternalAccessible := 'False'; ExternalVisible := 'False'; ExternalWritable := 'False'} : Bool;   //  TRUE if power supply 6 is OK
      ix_PowerSupply_Infeed_6 { ExternalAccessible := 'False'; ExternalVisible := 'False'; ExternalWritable := 'False'} : Bool;   //  400V power supply 6 infeed
      ix_PowerSupplyOk_7 { ExternalAccessible := 'False'; ExternalVisible := 'False'; ExternalWritable := 'False'} : Bool;   //  TRUE if power supply 7 is OK
      ix_PowerSupply_Infeed_7 { ExternalAccessible := 'False'; ExternalVisible := 'False'; ExternalWritable := 'False'} : Bool;   //  400V power supply 7 infeed
      ix_PowerSupplyOk_8 { ExternalAccessible := 'False'; ExternalVisible := 'False'; ExternalWritable := 'False'} : Bool;   //  TRUE if power supply 8 is OK
      ix_PowerSupply_Infeed_8 { ExternalAccessible := 'False'; ExternalVisible := 'False'; ExternalWritable := 'False'} : Bool;   //  400V power supply 8 infeed
      ix_PowerSupplyOk_9 { ExternalAccessible := 'False'; ExternalVisible := 'False'; ExternalWritable := 'False'} : Bool;   //  TRUE if power supply 9 is OK
      ix_PowerSupply_Infeed_9 { ExternalAccessible := 'False'; ExternalVisible := 'False'; ExternalWritable := 'False'} : Bool;   //  400V power supply 9 infeed
      ix_PowerSupplyOk_10 { ExternalAccessible := 'False'; ExternalVisible := 'False'; ExternalWritable := 'False'} : Bool;   //  TRUE if power supply 10 is OK
      ix_PowerSupply_Infeed_10 { ExternalAccessible := 'False'; ExternalVisible := 'False'; ExternalWritable := 'False'} : Bool;   //  400V power supply 10 infeed
      ix_HardwareOk { ExternalAccessible := 'False'; ExternalVisible := 'False'; ExternalWritable := 'False'} : Bool;   // TRUE when hardware is Ok
   END_VAR

   VAR_OUTPUT
      qUDT_HMIStatus { ExternalAccessible := 'False'; ExternalVisible := 'False'; ExternalWritable := 'False'} : "UDT_ControlPowerGroupStatus";   //  HMI status structure
      qUDT_Status { ExternalAccessible := 'False'; ExternalVisible := 'False'; ExternalWritable := 'False'} : "UDT_CommonStatus";   //  Common status structure
   END_VAR

   VAR_IN_OUT
      iqUDT_EquipmentControl : "UDT_EquipmentControl";   //  CIP Equipment control
      iqUDT_Statistics : "UDT_ControlPowerGroupStatistics";   //  CPG Statistics structure
   END_VAR

   VAR
      sUDT_HMIStatus { ExternalAccessible := 'False'; ExternalVisible := 'False'; ExternalWritable := 'False'; S7_SetPoint := 'False'} : "UDT_ControlPowerGroupStatus";   //  HMI status structure
      sUDT_CommonStatus { ExternalAccessible := 'False'; ExternalVisible := 'False'; ExternalWritable := 'False'; S7_SetPoint := 'False'} : "UDT_CommonStatus";   //  Common status structure
      sUDT_CommonStatusOld { ExternalAccessible := 'False'; ExternalVisible := 'False'; ExternalWritable := 'False'; S7_SetPoint := 'False'} : "UDT_CommonStatus";   //  Auxiliary status structure
      R_Trig_Warning {InstructionName := 'R_TRIG'; LibVersion := '1.0'; ExternalAccessible := 'False'; ExternalVisible := 'False'; ExternalWritable := 'False'; S7_SetPoint := 'False'} : R_TRIG;   //  Rising edge for warning
      R_Trig_Error {InstructionName := 'R_TRIG'; LibVersion := '1.0'; ExternalAccessible := 'False'; ExternalVisible := 'False'; ExternalWritable := 'False'; S7_SetPoint := 'False'} : R_TRIG;   //  Rising edge for error
      sw_NumberOfFailsAux { ExternalAccessible := 'False'; ExternalVisible := 'False'; ExternalWritable := 'False'} : Word;   //  Auxilary number of fails
      si_NumberOfFails { ExternalAccessible := 'False'; ExternalVisible := 'False'; ExternalWritable := 'False'} : Int;   //  Number of fails
      sx_WarningAux { ExternalAccessible := 'False'; ExternalVisible := 'False'; ExternalWritable := 'False'} : Bool;   //  Auxilary warninig
      sx_ErrorAux { ExternalAccessible := 'False'; ExternalVisible := 'False'; ExternalWritable := 'False'} : Bool;   //  Auxilary error
   END_VAR


BEGIN
	(*
	----------------------------------------------------------------------------------------

	Version history:
	Date        | Version   | Author        | Remark
	----------------------------------------------------------------------------------------
	03/10/2019  | 2.0       | C.Leite       | first release TIA 15.1
	15/10/2019  | 2.1       | L.Klar        | Updated status structure
	15/10/2019  | 2.2       | C. Leite      | UDTs and comments update
	17/10/2019  | 2.3       | S. Deulkar    | Added comments to interface signals
	04/11/2019  | 2.4       | C. Leite      | Power supplu 400V infeed state added
	12/11/2019  | 3.0       | P.Majka       | 3.0 MHS library release TIA 15.1
	04/12/2019  | 3.1       | C.Leite       | Remove number of power supplies input from interface
	25/02/2020  | 3.2       | S. Deulkar    | Modified to update ststus output every cycle
	09/07/2020  | 3.3       | S.Theocharis  | Bug fix in status update. Initialize static status instead output status
	21/02/2023  | 4.0       | F.Baten       | 4.0 Release TIA 17.5
	*)

	REGION 1 - Power Supply monitoring

